      ;ENDFOLD
      ;FOLD -- RSK Fehlerausgabe KF1 Initiator/Motor -- ;%{SE}%MKUKATPVW %CVW_COM %VCOMMENT %P 2:-- RSK Fehlerausgabe KF1 Initiator/Motor --, 3: VW_COMMENT
      ;ENDFOLD
      ;FOLD F322 = !F313 ;%{SE}%MKUKATPVW %CVW_SPS %VBOASG %P 2:F322 = !F313, 3: BOASG
         $FLAG[322] = NOT $FLAG[313]
      ;ENDFOLD
      ;FOLD -- Fraesfehler -- ;%{SE}%MKUKATPVW %CVW_COM %VCOMMENT %P 2:-- Fraesfehler --, 3: VW_COMMENT
      ;ENDFOLD
      ;FOLD F329 = F324 + F322 ;%{SE}%MKUKATPVW %CVW_SPS %VBOASG %P 2:F329 = F324 + F322, 3: BOASG
         $FLAG[329] = $FLAG[324] OR $FLAG[322]
      ;ENDFOLD
      ;FOLD -- Fraeser aus bei Fehler -- ;%{SE}%MKUKATPVW %CVW_COM %VCOMMENT %P 2:-- Fraeser aus bei Fehler --, 3: VW_COMMENT
      ;ENDFOLD
      ;FOLD A864 = !F329 ;%{SE}%MKUKATPVW %CVW_SPS %VBOASG %P 2:A864 = !F329, 3: BOASG
         $OUT[864] = NOT $FLAG[329]
      ;ENDFOLD
      ;FOLD -- Warte Fraesen fertig oder Timeout -- ;%{SE}%MKUKATPVW %CVW_COM %VCOMMENT %P 2:-- Warte Fraesen fertig oder Timeout --, 3: VW_COMMENT
      ;ENDFOLD
      ;FOLD Schritt 124 = (F79 & F98 + F78 & F94 & !F287 + T7) & A4039 ;%{SE}%MKUKATPVW %CVW_SPS %VST_CON %P 2:Schritt 124 = (F79 & F98 + F78 & F94 & !F287 + T7) & A4039, 3: ST_CON
         IF ($FLAG[79] AND $FLAG[98] OR $FLAG[78] AND $FLAG[94] AND NOT $FLAG[287] OR $TIMER_FLAG[7]) AND $OUT[4039] THEN
            PREVSTEP = $APP_INT[5]
            $APP_INT[5] = 124
         ENDIF
      ;ENDFOLD
      ;FOLD Schritt 124 = (F78 & F96 & F287 + T7) & A4039 ;%{SE}%MKUKATPVW %CVW_SPS %VST_CON %P 2:Schritt 124 = (F78 & F96 & F287 + T7) & A4039, 3: ST_CON
         IF ($FLAG[78] AND $FLAG[96] AND $FLAG[287] OR $TIMER_FLAG[7]) AND $OUT[4039] THEN
            PREVSTEP = $APP_INT[5]
            $APP_INT[5] = 124
         ENDIF
      ;ENDFOLD
   ;ENDFOLD
   ;FOLD SCHRITT 124 -- ROB STP1 SZ1 -- ;%{P}%MKUKATPVW,%CSTEP,%VST_NR,%P 1:SCHRITT, 2:124, 3: ROB STP1 SZ1
      ;FOLD ;%{H}
         Case 124
      ;ENDFOLD
      ;FOLD -- Hilfsflag SK Programmwechsel -- ;%{SE}%MKUKATPVW %CVW_COM %VCOMMENT %P 2:-- Hilfsflag SK Programmwechsel --, 3: VW_COMMENT
      ;ENDFOLD
      ;FOLD F334 = AUS ;%{SE}%MKUKATPVW %CVW_SPS %VBOASG %P 2:F334 = AUS, 3: BOASG
         $FLAG[334] = FALSE
      ;ENDFOLD
      ;FOLD -- KF1 runterfahren -- ;%{SE}%MKUKATPVW %CVW_COM %VCOMMENT %P 2:-- KF1 runterfahren --, 3: VW_COMMENT
      ;ENDFOLD
      ;FOLD A863 = AUS ;%{SE}%MKUKATPVW %CVW_SPS %VBOASG %P 2:A863 = AUS, 3: BOASG
         $OUT[863] = FALSE
      ;ENDFOLD
      ;FOLD -- Fraesfehler -- ;%{SE}%MKUKATPVW %CVW_COM %VCOMMENT %P 2:-- Fraesfehler --, 3: VW_COMMENT
      ;ENDFOLD
      ;FOLD F329 = T7 + F324 ;%{SE}%MKUKATPVW %CVW_SPS %VBOASG %P 2:F329 = T7 + F324, 3: BOASG
         $FLAG[329] = $TIMER_FLAG[7] OR $FLAG[324]
      ;ENDFOLD
      ;FOLD -- Hilfsflag Startfraesen -- ;%{SE}%MKUKATPVW %CVW_COM %VCOMMENT %P 2:-- Hilfsflag Startfraesen --, 3: VW_COMMENT
      ;ENDFOLD
      ;FOLD F96 = F96 & F287 ;%{SE}%MKUKATPVW %CVW_SPS %VBOASG %P 2:F96 = F96 & F287, 3: BOASG
         $FLAG[96] = $FLAG[96] AND $FLAG[287]
      ;ENDFOLD
      ;FOLD F287 = F78 ;%{SE}%MKUKATPVW %CVW_SPS %VBOASG %P 2:F287 = F78, 3: BOASG
         $FLAG[287] = $FLAG[78]
      ;ENDFOLD
      ;FOLD -- Wiederholung beim Startfraesen -- ;%{SE}%MKUKATPVW %CVW_COM %VCOMMENT %P 2:-- Wiederholung beim Startfraesen --, 3: VW_COMMENT
      ;ENDFOLD
      ;FOLD Schritt 121 = E863 & F78 & !F96 & !F329 & A4039 ;%{SE}%MKUKATPVW %CVW_SPS %VST_CON %P 2:Schritt 121 = E863 & F78 & !F96 & !F329 & A4039, 3: ST_CON
         IF $IN[863] AND $FLAG[78] AND NOT $FLAG[96] AND NOT $FLAG[329] AND $OUT[4039] THEN
            PREVSTEP = $APP_INT[5]
            $APP_INT[5] = 121
         ENDIF
      ;ENDFOLD
      ;FOLD -- Weiter wenn Fraesen fertig -- ;%{SE}%MKUKATPVW %CVW_COM %VCOMMENT %P 2:-- Weiter wenn Fraesen fertig --, 3: VW_COMMENT
      ;ENDFOLD
      ;FOLD Schritt 125 = E863 & (F79 & F98 + F78 & F96 + F329) & A4039 ;%{SE}%MKUKATPVW %CVW_SPS %VST_CON %P 2:Schritt 125 = E863 & (F79 & F98 + F78 & F96 + F329) & A4039, 3: ST_CON
         IF $IN[863] AND ($FLAG[79] AND $FLAG[98] OR $FLAG[78] AND $FLAG[96] OR $FLAG[329]) AND $OUT[4039] THEN
            PREVSTEP = $APP_INT[5]
            $APP_INT[5] = 125
         ENDIF
      ;ENDFOLD
      ;FOLD -- Weiter bei Fehler -- ;%{SE}%MKUKATPVW %CVW_COM %VCOMMENT %P 2:-- Weiter bei Fehler --, 3: VW_COMMENT
      ;ENDFOLD
      ;FOLD Schritt 127 = F329 & (E26 + E27) & A4039 ;%{SE}%MKUKATPVW %CVW_SPS %VST_CON %P 2:Schritt 127 = F329 & (E26 + E27) & A4039, 3: ST_CON
         IF $FLAG[329] AND ($IN[26] OR $IN[27]) AND $OUT[4039] THEN
            PREVSTEP = $APP_INT[5]
            $APP_INT[5] = 127
         ENDIF
      ;ENDFOLD
   ;ENDFOLD
   ;FOLD SCHRITT 125 -- ROB STP1 SZ1 -- ;%{P}%MKUKATPVW,%CSTEP,%VST_NR,%P 1:SCHRITT, 2:125, 3: ROB STP1 SZ1
      ;FOLD ;%{H}
         Case 125
      ;ENDFOLD
      ;FOLD -- KF1 einschalten -- ;%{SE}%MKUKATPVW %CVW_COM %VCOMMENT %P 2:-- KF1 einschalten --, 3: VW_COMMENT
      ;ENDFOLD
      ;FOLD A864 = AUS ;%{SE}%MKUKATPVW %CVW_SPS %VBOASG %P 2:A864 = AUS, 3: BOASG
         $OUT[864] = FALSE
      ;ENDFOLD
      ;FOLD bin3 (!F329) = 1 ;%{SE}%MKUKATPVW %CVW_SPS %VARIASG %P 2:bin3 (!F329) = 1, 3: ARIASG
         VW(#BINOUT,NOT $FLAG[329],3,1)
      ;ENDFOLD
      ;FOLD -- Wartezeit Programmwechsel SK -- ;%{SE}%MKUKATPVW %CVW_COM %VCOMMENT %P 2:-- Wartezeit Programmwechsel SK --, 3: VW_COMMENT
      ;ENDFOLD
      ;FOLD T8 ( !F334 ) = -2[1/10Sek] ;%{SE}%MKUKATPVW %CVW_SPS %VTASG %P 2:T8 ( !F334 ) = -2[1/10Sek], 3: TASG
         VW(#SET_TIME,NOT $FLAG[334],8,0,-2)
      ;ENDFOLD
      ;FOLD -- Hilfsflag SK Programmwechsel -- ;%{SE}%MKUKATPVW %CVW_COM %VCOMMENT %P 2:-- Hilfsflag SK Programmwechsel --, 3: VW_COMMENT
      ;ENDFOLD
      ;FOLD F334 = EIN ;%{SE}%MKUKATPVW %CVW_SPS %VBOASG %P 2:F334 = EIN, 3: BOASG
         $FLAG[334] = TRUE
      ;ENDFOLD
      ;FOLD Schritt 126 = T8 & A4039 ;%{SE}%MKUKATPVW %CVW_SPS %VST_CON %P 2:Schritt 126 = T8 & A4039, 3: ST_CON
         IF $TIMER_FLAG[8] AND $OUT[4039] THEN
            PREVSTEP = $APP_INT[5]
            $APP_INT[5] = 126
         ENDIF
      ;ENDFOLD
   ;ENDFOLD
   ;FOLD SCHRITT 126 -- ROB STP1 SZ1 -- ;%{P}%MKUKATPVW,%CSTEP,%VST_NR,%P 1:SCHRITT, 2:126, 3: ROB STP1 SZ1
      ;FOLD ;%{H}
         Case 126
      ;ENDFOLD
      ;FOLD -- Hilfsflag SK Programmwechsel -- ;%{SE}%MKUKATPVW %CVW_COM %VCOMMENT %P 2:-- Hilfsflag SK Programmwechsel --, 3: VW_COMMENT
      ;ENDFOLD
      ;FOLD F334 = AUS ;%{SE}%MKUKATPVW %CVW_SPS %VBOASG %P 2:F334 = AUS, 3: BOASG
         $FLAG[334] = FALSE
      ;ENDFOLD
      ;FOLD -- RSK Sammelstoerung -- ;%{SE}%MKUKATPVW %CVW_COM %VCOMMENT %P 2:-- RSK Sammelstoerung --, 3: VW_COMMENT
      ;ENDFOLD
      ;FOLD F329 = T7 ;%{SE}%MKUKATPVW %CVW_SPS %VBOASG %P 2:F329 = T7, 3: BOASG
         $FLAG[329] = $TIMER_FLAG[7]
      ;ENDFOLD
      ;FOLD -- Quitt. Fraesen SK1 -- ;%{SE}%MKUKATPVW %CVW_COM %VCOMMENT %P 2:-- Quitt. Fraesen SK1 --, 3: VW_COMMENT
      ;ENDFOLD
      ;FOLD A786 = !F329 & !F322 ;%{SE}%MKUKATPVW %CVW_SPS %VBOASG %P 2:A786 = !F329 & !F322, 3: BOASG
         $OUT[786] = NOT $FLAG[329] AND NOT $FLAG[322]
      ;ENDFOLD
      ;FOLD Schritt 127 = !E786 & E787 & !E788 & !F329 ;%{SE}%MKUKATPVW %CVW_SPS %VST_CON %P 2:Schritt 127 = !E786 & E787 & !E788 & !F329, 3: ST_CON
         IF NOT $IN[786] AND $IN[787] AND NOT $IN[788] AND NOT $FLAG[329] THEN
            PREVSTEP = $APP_INT[5]
            $APP_INT[5] = 127
         ENDIF
      ;ENDFOLD
   ;ENDFOLD
   ;FOLD SCHRITT 127 -- ROB STP1 SZ1 # Ende -- ;%{P}%MKUKATPVW,%CSTEP,%VST_NR,%P 1:SCHRITT, 2:127, 3: ROB STP1 SZ1 # Ende
      ;FOLD ;%{H}
         Case 127
      ;ENDFOLD
      ;FOLD -- RSK Sammelstoerung -- ;%{SE}%MKUKATPVW %CVW_COM %VCOMMENT %P 2:-- RSK Sammelstoerung --, 3: VW_COMMENT
      ;ENDFOLD
      ;FOLD F329 = T7 ;%{SE}%MKUKATPVW %CVW_SPS %VBOASG %P 2:F329 = T7, 3: BOASG
         $FLAG[329] = $TIMER_FLAG[7]
      ;ENDFOLD
      ;FOLD F91 = !F329 ;%{SE}%MKUKATPVW %CVW_SPS %VBOASG %P 2:F91 = !F329, 3: BOASG
         $FLAG[91] = NOT $FLAG[329]
      ;ENDFOLD
      ;FOLD Schritt 120 = F329 & (E26 + E27) & A4039 ;%{SE}%MKUKATPVW %CVW_SPS %VST_CON %P 2:Schritt 120 = F329 & (E26 + E27) & A4039, 3: ST_CON
         IF $FLAG[329] AND ($IN[26] OR $IN[27]) AND $OUT[4039] THEN
            PREVSTEP = $APP_INT[5]
            $APP_INT[5] = 120
         ENDIF
      ;ENDFOLD
      ;FOLD Schritt 1 = F91 & !F329 & A4039 ;%{SE}%MKUKATPVW %CVW_SPS %VST_CON %P 2:Schritt 1 = F91 & !F329 & A4039, 3: ST_CON
         IF $FLAG[91] AND NOT $FLAG[329] AND $OUT[4039] THEN
            PREVSTEP = $APP_INT[5]
            $APP_INT[5] = 1
         ENDIF
      ;ENDFOLD
   ;ENDFOLD
   ;FOLD SCHRITT 128 -- MS1 Reinigung (an KS3)-- ;%{P}%MKUKATPVW,%CSTEP,%VST_NR,%P 1:SCHRITT, 2:128, 3: MS1 Reinigung (an KS3)
      ;FOLD ;%{H}
         Case 128
      ;ENDFOLD
      ;FOLD -- RSK gestartet -- ;%{SE}%MKUKATPVW %CVW_COM %VCOMMENT %P 2:-- RSK gestartet --, 3: VW_COMMENT
      ;ENDFOLD
      ;FOLD F321 = AUS ;%{SE}%MKUKATPVW %CVW_SPS %VBOASG %P 2:F321 = AUS, 3: BOASG
         $FLAG[321] = FALSE
      ;ENDFOLD
      ;FOLD F323 = AUS ;%{SE}%MKUKATPVW %CVW_SPS %VBOASG %P 2:F323 = AUS, 3: BOASG
         $FLAG[323] = FALSE
      ;ENDFOLD
      ;FOLD F324 = AUS ;%{SE}%MKUKATPVW %CVW_SPS %VBOASG %P 2:F324 = AUS, 3: BOASG
         $FLAG[324] = FALSE
      ;ENDFOLD
      ;FOLD F329 = AUS ;%{SE}%MKUKATPVW %CVW_SPS %VBOASG %P 2:F329 = AUS, 3: BOASG
         $FLAG[329] = FALSE
      ;ENDFOLD
      ;FOLD -- MS1 Reinigung gestartet -- ;%{SE}%MKUKATPVW %CVW_COM %VCOMMENT %P 2:-- MS1 Reinigung gestartet --, 3: VW_COMMENT
      ;ENDFOLD
      ;FOLD F604 = EIN ;%{SE}%MKUKATPVW %CVW_SPS %VBOASG %P 2:F604 = EIN, 3: BOASG
         $FLAG[604] = TRUE
      ;ENDFOLD
      ;FOLD -- Ueberwachungszeit KS3 schwenken -- ;%{SE}%MKUKATPVW %CVW_COM %VCOMMENT %P 2:-- Ueberwachungszeit KS3 schwenken --, 3: VW_COMMENT
      ;ENDFOLD
      ;FOLD t8 ( EIN ) = -100[1/10Sek] ;%{SE}%MKUKATPVW %CVW_SPS %VTASG %P 2:t8 ( EIN ) = -100[1/10Sek], 3: TASG
         VW(#SET_TIME,TRUE,8,0,-100)
      ;ENDFOLD
      ;FOLD Schritt 129 = A4039 ;%{SE}%MKUKATPVW %CVW_SPS %VST_CON %P 2:Schritt 129 = A4039, 3: ST_CON
         IF $OUT[4039] THEN
            PREVSTEP = $APP_INT[5]
            $APP_INT[5] = 129
         ENDIF
      ;ENDFOLD
   ;ENDFOLD
   ;FOLD SCHRITT 129 -- MS1 Reinigung (an KS3) -- ;%{P}%MKUKATPVW,%CSTEP,%VST_NR,%P 1:SCHRITT, 2:129, 3: MS1 Reinigung (an KS3)
      ;FOLD ;%{H}
         Case 129
      ;ENDFOLD
      ;FOLD -- RSK Fehlerausgabe KS3 Ruhest. -- ;%{SE}%MKUKATPVW %CVW_COM %VCOMMENT %P 2:-- RSK Fehlerausgabe KS3 Ruhest. --, 3: VW_COMMENT
      ;ENDFOLD
      ;FOLD F323 = !E1156 ;%{SE}%MKUKATPVW %CVW_SPS %VBOASG %P 2:F323 = !E1156, 3: BOASG
         $FLAG[323] = NOT $IN[1156]
      ;ENDFOLD
      ;FOLD -- RSK Sammelstoerung -- ;%{SE}%MKUKATPVW %CVW_COM %VCOMMENT %P 2:-- RSK Sammelstoerung --, 3: VW_COMMENT
      ;ENDFOLD
      ;FOLD F329 = F323 ;%{SE}%MKUKATPVW %CVW_SPS %VBOASG %P 2:F329 = F323, 3: BOASG
         $FLAG[329] = $FLAG[323]
      ;ENDFOLD
      ;FOLD Schritt 128 = (E26 + E27) & F323 & A4039 ;%{SE}%MKUKATPVW %CVW_SPS %VST_CON %P 2:Schritt 128 = (E26 + E27) & F323 & A4039, 3: ST_CON
         IF ($IN[26] OR $IN[27]) AND $FLAG[323] AND $OUT[4039] THEN
            PREVSTEP = $APP_INT[5]
            $APP_INT[5] = 128
         ENDIF
      ;ENDFOLD
      ;FOLD Schritt 130 = (!F323 + T8) & A4039 ;%{SE}%MKUKATPVW %CVW_SPS %VST_CON %P 2:Schritt 130 = (!F323 + T8) & A4039, 3: ST_CON
         IF (NOT $FLAG[323] OR $TIMER_FLAG[8]) AND $OUT[4039] THEN
            PREVSTEP = $APP_INT[5]
            $APP_INT[5] = 130
         ENDIF
      ;ENDFOLD
   ;ENDFOLD
   ;FOLD SCHRITT 130 -- MS1 Reinigung (an KS3) -- ;%{P}%MKUKATPVW,%CSTEP,%VST_NR,%P 1:SCHRITT, 2:130, 3: MS1 Reinigung (an KS3)
      ;FOLD ;%{H}
         Case 130
      ;ENDFOLD
      ;FOLD -- KS3 in Arbeitsstellung schwenken -- ;%{SE}%MKUKATPVW %CVW_COM %VCOMMENT %P 2:-- KS3 in Arbeitsstellung schwenken --, 3: VW_COMMENT
      ;ENDFOLD
      ;FOLD A1160 = !E1157 ;%{SE}%MKUKATPVW %CVW_SPS %VBOASG %P 2:A1160 = !E1157, 3: BOASG
         $OUT[1160] = NOT $IN[1157]
      ;ENDFOLD
      ;FOLD Schritt 131 = A4039 ;%{SE}%MKUKATPVW %CVW_SPS %VST_CON %P 2:Schritt 131 = A4039, 3: ST_CON
         IF $OUT[4039] THEN
            PREVSTEP = $APP_INT[5]
            $APP_INT[5] = 131
         ENDIF
      ;ENDFOLD
   ;ENDFOLD
   ;FOLD SCHRITT 131 -- MS1 Reinigung (an KS3) -- ;%{P}%MKUKATPVW,%CSTEP,%VST_NR,%P 1:SCHRITT, 2:131, 3: MS1 Reinigung (an KS3)
      ;FOLD ;%{H}
         Case 131
      ;ENDFOLD
      ;FOLD -- RSK Fehlerausgabe KS3 Arbeitsstellung -- ;%{SE}%MKUKATPVW %CVW_COM %VCOMMENT %P 2:-- RSK Fehlerausgabe KS3 Arbeitsstellung --, 3: VW_COMMENT
      ;ENDFOLD
      ;FOLD F324 = !E1157 & T8 + F324 ;%{SE}%MKUKATPVW %CVW_SPS %VBOASG %P 2:F324 = !E1157 & T8 + F324, 3: BOASG
         $FLAG[324] = NOT $IN[1157] AND $TIMER_FLAG[8] OR $FLAG[324]
      ;ENDFOLD
      ;FOLD -- RSK Sammelstoerung -- ;%{SE}%MKUKATPVW %CVW_COM %VCOMMENT %P 2:-- RSK Sammelstoerung --, 3: VW_COMMENT
      ;ENDFOLD
      ;FOLD F329 = F324 ;%{SE}%MKUKATPVW %CVW_SPS %VBOASG %P 2:F329 = F324, 3: BOASG
         $FLAG[329] = $FLAG[324]
      ;ENDFOLD
      ;FOLD Schritt 128 = F324 & (E26 + E27) & A4039 ;%{SE}%MKUKATPVW %CVW_SPS %VST_CON %P 2:Schritt 128 = F324 & (E26 + E27) & A4039, 3: ST_CON
         IF $FLAG[324] AND ($IN[26] OR $IN[27]) AND $OUT[4039] THEN
            PREVSTEP = $APP_INT[5]
            $APP_INT[5] = 128
         ENDIF
      ;ENDFOLD
      ;FOLD Schritt 132 = !F324 & E1157 & !E1159 & A4039 ;%{SE}%MKUKATPVW %CVW_SPS %VST_CON %P 2:Schritt 132 = !F324 & E1157 & !E1159 & A4039, 3: ST_CON
         IF NOT $FLAG[324] AND $IN[1157] AND NOT $IN[1159] AND $OUT[4039] THEN
            PREVSTEP = $APP_INT[5]
            $APP_INT[5] = 132
         ENDIF
      ;ENDFOLD
   ;ENDFOLD
   ;FOLD SCHRITT 132 -- MS1 Reinigung (an KS3) -- ;%{P}%MKUKATPVW,%CSTEP,%VST_NR,%P 1:SCHRITT, 2:132, 3: MS1 Reinigung (an KS3)
      ;FOLD ;%{H}
         Case 132
      ;ENDFOLD
      ;FOLD A1864 = AUS ;%{SE}%MKUKATPVW %CVW_SPS %VBOASG %P 2:A1864 = AUS, 3: BOASG
         $OUT[1864] = FALSE
      ;ENDFOLD
      ;FOLD A2168 = AUS ;%{SE}%MKUKATPVW %CVW_SPS %VBOASG %P 2:A2168 = AUS, 3: BOASG
         $OUT[2168] = FALSE
      ;ENDFOLD
      ;FOLD -- Ueberwachungszeit Versetzeinheit -- ;%{SE}%MKUKATPVW %CVW_COM %VCOMMENT %P 2:-- Ueberwachungszeit Versetzeinheit --, 3: VW_COMMENT
      ;ENDFOLD
      ;FOLD t8 ( EIN ) = -50[1/10Sek] ;%{SE}%MKUKATPVW %CVW_SPS %VTASG %P 2:t8 ( EIN ) = -50[1/10Sek], 3: TASG
         VW(#SET_TIME,TRUE,8,0,-50)
      ;ENDFOLD
      ;FOLD -- Ueberwachungszeit Reinigung -- ;%{SE}%MKUKATPVW %CVW_COM %VCOMMENT %P 2:-- Ueberwachungszeit Reinigung --, 3: VW_COMMENT
      ;ENDFOLD
      ;FOLD t9 ( EIN ) = -80[1/10Sek] ;%{SE}%MKUKATPVW %CVW_SPS %VTASG %P 2:t9 ( EIN ) = -80[1/10Sek], 3: TASG
         VW(#SET_TIME,TRUE,9,0,-80)
      ;ENDFOLD
      ;FOLD Schritt 133 = A4039 ;%{SE}%MKUKATPVW %CVW_SPS %VST_CON %P 2:Schritt 133 = A4039, 3: ST_CON
         IF $OUT[4039] THEN
            PREVSTEP = $APP_INT[5]
            $APP_INT[5] = 133
         ENDIF
      ;ENDFOLD
   ;ENDFOLD
   ;FOLD SCHRITT 133 -- MS1 Reinigung (an KS3) -- ;%{P}%MKUKATPVW,%CSTEP,%VST_NR,%P 1:SCHRITT, 2:133, 3: MS1 Reinigung (an KS3)
      ;FOLD ;%{H}
         Case 133
      ;ENDFOLD
      ;FOLD -- RSK Fehlerausgabe Versetzeinheit -- ;%{SE}%MKUKATPVW %CVW_COM %VCOMMENT %P 2:-- RSK Fehlerausgabe Versetzeinheit --, 3: VW_COMMENT
      ;ENDFOLD
      ;FOLD F328 = F576 & T8 ;%{SE}%MKUKATPVW %CVW_SPS %VBOASG %P 2:F328 = F576 & T8, 3: BOASG
         $FLAG[328] = $FLAG[576] AND $TIMER_FLAG[8]
      ;ENDFOLD
      ;FOLD -- RSK Sammelstoerung -- ;%{SE}%MKUKATPVW %CVW_COM %VCOMMENT %P 2:-- RSK Sammelstoerung --, 3: VW_COMMENT
      ;ENDFOLD
      ;FOLD F329 = T8 ;%{SE}%MKUKATPVW %CVW_SPS %VBOASG %P 2:F329 = T8, 3: BOASG
         $FLAG[329] = $TIMER_FLAG[8]
      ;ENDFOLD
      ;FOLD -- Versetzeinheit in Arbeitsst. schw. -- ;%{SE}%MKUKATPVW %CVW_COM %VCOMMENT %P 2:-- Versetzeinheit in Arbeitsst. schw. --, 3: VW_COMMENT
      ;ENDFOLD
      ;FOLD A2168 = !E2168 & F576 ;%{SE}%MKUKATPVW %CVW_SPS %VBOASG %P 2:A2168 = !E2168 & F576, 3: BOASG
         $OUT[2168] = NOT $IN[2168] AND $FLAG[576]
      ;ENDFOLD
      ;FOLD Schritt 132 = A2168 & T8 & (E26 + E27) & A4039 ;%{SE}%MKUKATPVW %CVW_SPS %VST_CON %P 2:Schritt 132 = A2168 & T8 & (E26 + E27) & A4039, 3: ST_CON
         IF $OUT[2168] AND $TIMER_FLAG[8] AND ($IN[26] OR $IN[27]) AND $OUT[4039] THEN
            PREVSTEP = $APP_INT[5]
            $APP_INT[5] = 132
         ENDIF
      ;ENDFOLD
      ;FOLD Schritt 134 = (E2168 & F576 + !E2168 & !F576) & A4039 ;%{SE}%MKUKATPVW %CVW_SPS %VST_CON %P 2:Schritt 134 = (E2168 & F576 + !E2168 & !F576) & A4039, 3: ST_CON
         IF ($IN[2168] AND $FLAG[576] OR NOT $IN[2168] AND NOT $FLAG[576]) AND $OUT[4039] THEN
            PREVSTEP = $APP_INT[5]
            $APP_INT[5] = 134
         ENDIF
      ;ENDFOLD
   ;ENDFOLD
   ;FOLD SCHRITT 134 -- MS1 Reinigung (an KS3) -- ;%{P}%MKUKATPVW,%CSTEP,%VST_NR,%P 1:SCHRITT, 2:134, 3: MS1 Reinigung (an KS3)
      ;FOLD ;%{H}
         Case 134
      ;ENDFOLD
      ;FOLD -- RSK Sammelstoerung -- ;%{SE}%MKUKATPVW %CVW_COM %VCOMMENT %P 2:-- RSK Sammelstoerung --, 3: VW_COMMENT
      ;ENDFOLD
      ;FOLD F329 = T9 ;%{SE}%MKUKATPVW %CVW_SPS %VBOASG %P 2:F329 = T9, 3: BOASG
         $FLAG[329] = $TIMER_FLAG[9]
      ;ENDFOLD
      ;FOLD -- MS1 Ausblasen EIN -- ;%{SE}%MKUKATPVW %CVW_COM %VCOMMENT %P 2:-- MS1 Ausblasen EIN --, 3: VW_COMMENT
      ;ENDFOLD
      ;FOLD A1870 = EIN ;%{SE}%MKUKATPVW %CVW_SPS %VBOASG %P 2:A1870 = EIN, 3: BOASG
         $OUT[1870] = TRUE
      ;ENDFOLD
      ;FOLD -- MS1 Reinigung starten -- ;%{SE}%MKUKATPVW %CVW_COM %VCOMMENT %P 2:-- MS1 Reinigung starten --, 3: VW_COMMENT
      ;ENDFOLD
      ;FOLD A1864 = EIN ;%{SE}%MKUKATPVW %CVW_SPS %VBOASG %P 2:A1864 = EIN, 3: BOASG
         $OUT[1864] = TRUE
      ;ENDFOLD
      ;FOLD Schritt 132 = !E1864 & T9 & (E26 + E27) & A4039 ;%{SE}%MKUKATPVW %CVW_SPS %VST_CON %P 2:Schritt 132 = !E1864 & T9 & (E26 + E27) & A4039, 3: ST_CON
         IF NOT $IN[1864] AND $TIMER_FLAG[9] AND ($IN[26] OR $IN[27]) AND $OUT[4039] THEN
            PREVSTEP = $APP_INT[5]
            $APP_INT[5] = 132
         ENDIF
      ;ENDFOLD
      ;FOLD Schritt 135 = E1864 & A4039 ;%{SE}%MKUKATPVW %CVW_SPS %VST_CON %P 2:Schritt 135 = E1864 & A4039, 3: ST_CON
         IF $IN[1864] AND $OUT[4039] THEN
            PREVSTEP = $APP_INT[5]
            $APP_INT[5] = 135
         ENDIF
      ;ENDFOLD
   ;ENDFOLD
   ;FOLD SCHRITT 135 -- MS1 Reinigung (an KS3) -- ;%{P}%MKUKATPVW,%CSTEP,%VST_NR,%P 1:SCHRITT, 2:135, 3: MS1 Reinigung (an KS3)
      ;FOLD ;%{H}
         Case 135
      ;ENDFOLD
      ;FOLD -- MS1 Reinigung beenden -- ;%{SE}%MKUKATPVW %CVW_COM %VCOMMENT %P 2:-- MS1 Reinigung beenden --, 3: VW_COMMENT
      ;ENDFOLD
      ;FOLD A1864 = AUS ;%{SE}%MKUKATPVW %CVW_SPS %VBOASG %P 2:A1864 = AUS, 3: BOASG
         $OUT[1864] = FALSE
      ;ENDFOLD
      ;FOLD -- MS1 Ausblasen AUS -- ;%{SE}%MKUKATPVW %CVW_COM %VCOMMENT %P 2:-- MS1 Ausblasen AUS --, 3: VW_COMMENT
      ;ENDFOLD
      ;FOLD A1870 = AUS ;%{SE}%MKUKATPVW %CVW_SPS %VBOASG %P 2:A1870 = AUS, 3: BOASG
         $OUT[1870] = FALSE
      ;ENDFOLD
      ;FOLD -- MS1 Einspruehen EIN -- ;%{SE}%MKUKATPVW %CVW_COM %VCOMMENT %P 2:-- MS1 Einspruehen EIN --, 3: VW_COMMENT
      ;ENDFOLD
      ;FOLD A520 = !F574 & F575 ;%{SE}%MKUKATPVW %CVW_SPS %VBOASG %P 2:A520 = !F574 & F575, 3: BOASG
         $OUT[520] = NOT $FLAG[574] AND $FLAG[575]
      ;ENDFOLD
      ;FOLD A1871 = F574 & F575 ;%{SE}%MKUKATPVW %CVW_SPS %VBOASG %P 2:A1871 = F574 & F575, 3: BOASG
         $OUT[1871] = $FLAG[574] AND $FLAG[575]
      ;ENDFOLD
      ;FOLD -- Einschaltdauer Einspruehen -- ;%{SE}%MKUKATPVW %CVW_COM %VCOMMENT %P 2:-- Einschaltdauer Einspruehen --, 3: VW_COMMENT
      ;ENDFOLD
      ;FOLD t7 ( EIN ) = i23[1/10Sek] ;%{SE}%MKUKATPVW %CVW_SPS %VTASG %P 2:t7 ( EIN ) = i23[1/10Sek], 3: TASG
         VW(#SET_TIME,TRUE,7,0,$COUNT_I[23])
      ;ENDFOLD
      ;FOLD Schritt 136 = A4039 ;%{SE}%MKUKATPVW %CVW_SPS %VST_CON %P 2:Schritt 136 = A4039, 3: ST_CON
         IF $OUT[4039] THEN
            PREVSTEP = $APP_INT[5]
            $APP_INT[5] = 136
         ENDIF
      ;ENDFOLD
   ;ENDFOLD
   ;FOLD SCHRITT 136 -- MS1 Reinigung (an KS3) -- ;%{P}%MKUKATPVW,%CSTEP,%VST_NR,%P 1:SCHRITT, 2:136, 3: MS1 Reinigung (an KS3)
      ;FOLD ;%{H}
         Case 136
      ;ENDFOLD
      ;FOLD F323 = AUS ;%{SE}%MKUKATPVW %CVW_SPS %VBOASG %P 2:F323 = AUS, 3: BOASG
         $FLAG[323] = FALSE
      ;ENDFOLD
      ;FOLD -- Ueberwachungszeit KS3 schwenken -- ;%{SE}%MKUKATPVW %CVW_COM %VCOMMENT %P 2:-- Ueberwachungszeit KS3 schwenken --, 3: VW_COMMENT
      ;ENDFOLD
      ;FOLD t8 ( EIN ) = -100[1/10Sek] ;%{SE}%MKUKATPVW %CVW_SPS %VTASG %P 2:t8 ( EIN ) = -100[1/10Sek], 3: TASG
         VW(#SET_TIME,TRUE,8,0,-100)
      ;ENDFOLD
      ;FOLD Schritt 137 = T7 & A4039 ;%{SE}%MKUKATPVW %CVW_SPS %VST_CON %P 2:Schritt 137 = T7 & A4039, 3: ST_CON
         IF $TIMER_FLAG[7] AND $OUT[4039] THEN
            PREVSTEP = $APP_INT[5]
            $APP_INT[5] = 137
         ENDIF
      ;ENDFOLD
   ;ENDFOLD
   ;FOLD SCHRITT 137 -- MS1 Reinigung (an KS3) -- ;%{P}%MKUKATPVW,%CSTEP,%VST_NR,%P 1:SCHRITT, 2:137, 3: MS1 Reinigung (an KS3)
      ;FOLD ;%{H}
         Case 137
      ;ENDFOLD
      ;FOLD -- MS1 Einspruehen AUS -- ;%{SE}%MKUKATPVW %CVW_COM %VCOMMENT %P 2:-- MS1 Einspruehen AUS --, 3: VW_COMMENT
      ;ENDFOLD
      ;FOLD A520 = AUS ;%{SE}%MKUKATPVW %CVW_SPS %VBOASG %P 2:A520 = AUS, 3: BOASG
         $OUT[520] = FALSE
      ;ENDFOLD
      ;FOLD A1871 = AUS ;%{SE}%MKUKATPVW %CVW_SPS %VBOASG %P 2:A1871 = AUS, 3: BOASG
         $OUT[1871] = FALSE
      ;ENDFOLD
      ;FOLD -- RSK Fehlerausgabe KS3 Ruhest. -- ;%{SE}%MKUKATPVW %CVW_COM %VCOMMENT %P 2:-- RSK Fehlerausgabe KS3 Ruhest. --, 3: VW_COMMENT
      ;ENDFOLD
      ;FOLD F324 = !E1157 ;%{SE}%MKUKATPVW %CVW_SPS %VBOASG %P 2:F324 = !E1157, 3: BOASG
         $FLAG[324] = NOT $IN[1157]
      ;ENDFOLD
      ;FOLD -- RSK Sammelstoerung -- ;%{SE}%MKUKATPVW %CVW_COM %VCOMMENT %P 2:-- RSK Sammelstoerung --, 3: VW_COMMENT
      ;ENDFOLD
      ;FOLD F329 = F324 + T8 ;%{SE}%MKUKATPVW %CVW_SPS %VBOASG %P 2:F329 = F324 + T8, 3: BOASG
         $FLAG[329] = $FLAG[324] OR $TIMER_FLAG[8]
      ;ENDFOLD
      ;FOLD Schritt 136 = (E26 + E27) & F324 & A4039 ;%{SE}%MKUKATPVW %CVW_SPS %VST_CON %P 2:Schritt 136 = (E26 + E27) & F324 & A4039, 3: ST_CON
         IF ($IN[26] OR $IN[27]) AND $FLAG[324] AND $OUT[4039] THEN
            PREVSTEP = $APP_INT[5]
            $APP_INT[5] = 136
         ENDIF
      ;ENDFOLD
      ;FOLD Schritt 138 = (!F324 + T8) & A4039 ;%{SE}%MKUKATPVW %CVW_SPS %VST_CON %P 2:Schritt 138 = (!F324 + T8) & A4039, 3: ST_CON
         IF (NOT $FLAG[324] OR $TIMER_FLAG[8]) AND $OUT[4039] THEN
            PREVSTEP = $APP_INT[5]
            $APP_INT[5] = 138
         ENDIF
      ;ENDFOLD
   ;ENDFOLD
   ;FOLD SCHRITT 138 -- MS1 Reinigung (an KS3) -- ;%{P}%MKUKATPVW,%CSTEP,%VST_NR,%P 1:SCHRITT, 2:138, 3: MS1 Reinigung (an KS3)
      ;FOLD ;%{H}
         Case 138
      ;ENDFOLD
      ;FOLD -- KS3 in Ruhestellung schwenken -- ;%{SE}%MKUKATPVW %CVW_COM %VCOMMENT %P 2:-- KS3 in Ruhestellung schwenken --, 3: VW_COMMENT
      ;ENDFOLD
      ;FOLD A1160 = !E1156 ;%{SE}%MKUKATPVW %CVW_SPS %VBOASG %P 2:A1160 = !E1156, 3: BOASG
         $OUT[1160] = NOT $IN[1156]
      ;ENDFOLD
      ;FOLD Schritt 139 = A4039 ;%{SE}%MKUKATPVW %CVW_SPS %VST_CON %P 2:Schritt 139 = A4039, 3: ST_CON
         IF $OUT[4039] THEN
            PREVSTEP = $APP_INT[5]
            $APP_INT[5] = 139
         ENDIF
      ;ENDFOLD
   ;ENDFOLD
   ;FOLD SCHRITT 139 -- MS1 Reinigung (an KS3) -- ;%{P}%MKUKATPVW,%CSTEP,%VST_NR,%P 1:SCHRITT, 2:139, 3: MS1 Reinigung (an KS3)
      ;FOLD ;%{H}
         Case 139
      ;ENDFOLD
      ;FOLD -- RSK Fehlerausgabe KS3 Ruhestellung -- ;%{SE}%MKUKATPVW %CVW_COM %VCOMMENT %P 2:-- RSK Fehlerausgabe KS3 Ruhestellung --, 3: VW_COMMENT
      ;ENDFOLD
      ;FOLD F323 = !E1156 & T8 + F323 ;%{SE}%MKUKATPVW %CVW_SPS %VBOASG %P 2:F323 = !E1156 & T8 + F323, 3: BOASG
         $FLAG[323] = NOT $IN[1156] AND $TIMER_FLAG[8] OR $FLAG[323]
      ;ENDFOLD
      ;FOLD -- RSK Sammelstoerung -- ;%{SE}%MKUKATPVW %CVW_COM %VCOMMENT %P 2:-- RSK Sammelstoerung --, 3: VW_COMMENT
      ;ENDFOLD
      ;FOLD F329 = F323 ;%{SE}%MKUKATPVW %CVW_SPS %VBOASG %P 2:F329 = F323, 3: BOASG
         $FLAG[329] = $FLAG[323]
      ;ENDFOLD
      ;FOLD Schritt 136 = F323 & (E26 + E27) & A4039 ;%{SE}%MKUKATPVW %CVW_SPS %VST_CON %P 2:Schritt 136 = F323 & (E26 + E27) & A4039, 3: ST_CON
         IF $FLAG[323] AND ($IN[26] OR $IN[27]) AND $OUT[4039] THEN
            PREVSTEP = $APP_INT[5]
            $APP_INT[5] = 136
         ENDIF
      ;ENDFOLD
      ;FOLD Schritt 140 = E1156 & !E1158 & A4039 ;%{SE}%MKUKATPVW %CVW_SPS %VST_CON %P 2:Schritt 140 = E1156 & !E1158 & A4039, 3: ST_CON
         IF $IN[1156] AND NOT $IN[1158] AND $OUT[4039] THEN
            PREVSTEP = $APP_INT[5]
            $APP_INT[5] = 140
         ENDIF
      ;ENDFOLD
   ;ENDFOLD
   ;FOLD SCHRITT 140 -- MS1 Reinigung (an KS3) -- ;%{P}%MKUKATPVW,%CSTEP,%VST_NR,%P 1:SCHRITT, 2:140, 3: MS1 Reinigung (an KS3)
      ;FOLD ;%{H}
         Case 140
      ;ENDFOLD
      ;FOLD F323 = AUS ;%{SE}%MKUKATPVW %CVW_SPS %VBOASG %P 2:F323 = AUS, 3: BOASG
         $FLAG[323] = FALSE
      ;ENDFOLD
      ;FOLD F329 = AUS ;%{SE}%MKUKATPVW %CVW_SPS %VBOASG %P 2:F329 = AUS, 3: BOASG
         $FLAG[329] = FALSE
      ;ENDFOLD
      ;FOLD -- MS1 Zaehler ruecksetzen -- ;%{SE}%MKUKATPVW %CVW_COM %VCOMMENT %P 2:-- MS1 Zaehler ruecksetzen --, 3: VW_COMMENT
      ;ENDFOLD
      ;FOLD -- MS1 FRG Reinigung -- ;%{SE}%MKUKATPVW %CVW_COM %VCOMMENT %P 2:-- MS1 FRG Reinigung --, 3: VW_COMMENT
      ;ENDFOLD
      ;FOLD F603 = AUS ;%{SE}%MKUKATPVW %CVW_SPS %VBOASG %P 2:F603 = AUS, 3: BOASG
         $FLAG[603] = FALSE
      ;ENDFOLD
      ;FOLD -- MS1 Reinigung FK -- ;%{SE}%MKUKATPVW %CVW_COM %VCOMMENT %P 2:-- MS1 Reinigung FK --, 3: VW_COMMENT
      ;ENDFOLD
      ;FOLD F605 = EIN ;%{SE}%MKUKATPVW %CVW_SPS %VBOASG %P 2:F605 = EIN, 3: BOASG
         $FLAG[605] = TRUE
      ;ENDFOLD
      ;FOLD t8 ( EIN ) = STOP ;%{SE}%MKUKATPVW %CVW_SPS %VTSTOP %P 2:t8 ( EIN ) = STOP, 3: TSTOP
         VW(#SET_TIME,TRUE,8,1,0)
      ;ENDFOLD
      ;FOLD Schritt 1 = A4039 ;%{SE}%MKUKATPVW %CVW_SPS %VST_CON %P 2:Schritt 1 = A4039, 3: ST_CON
         IF $OUT[4039] THEN
            PREVSTEP = $APP_INT[5]
            $APP_INT[5] = 1
         ENDIF
      ;ENDFOLD
   ;ENDFOLD
   ;FOLD SCHRITT 141 -- MS2 Reinigung (an KS2) -- ;%{P}%MKUKATPVW,%CSTEP,%VST_NR,%P 1:SCHRITT, 2:141, 3: MS2 Reinigung (an KS2)
      ;FOLD ;%{H}
         Case 141
      ;ENDFOLD
      ;FOLD -- RSK gestartet -- ;%{SE}%MKUKATPVW %CVW_COM %VCOMMENT %P 2:-- RSK gestartet --, 3: VW_COMMENT
      ;ENDFOLD
      ;FOLD F321 = AUS ;%{SE}%MKUKATPVW %CVW_SPS %VBOASG %P 2:F321 = AUS, 3: BOASG
         $FLAG[321] = FALSE
      ;ENDFOLD
      ;FOLD F323 = AUS ;%{SE}%MKUKATPVW %CVW_SPS %VBOASG %P 2:F323 = AUS, 3: BOASG
         $FLAG[323] = FALSE
      ;ENDFOLD
      ;FOLD F324 = AUS ;%{SE}%MKUKATPVW %CVW_SPS %VBOASG %P 2:F324 = AUS, 3: BOASG
         $FLAG[324] = FALSE
      ;ENDFOLD
      ;FOLD F329 = AUS ;%{SE}%MKUKATPVW %CVW_SPS %VBOASG %P 2:F329 = AUS, 3: BOASG
         $FLAG[329] = FALSE
      ;ENDFOLD
      ;FOLD -- MS2 Reinigung gestartet -- ;%{SE}%MKUKATPVW %CVW_COM %VCOMMENT %P 2:-- MS2 Reinigung gestartet --, 3: VW_COMMENT
      ;ENDFOLD
      ;FOLD F608 = EIN ;%{SE}%MKUKATPVW %CVW_SPS %VBOASG %P 2:F608 = EIN, 3: BOASG
         $FLAG[608] = TRUE
      ;ENDFOLD
      ;FOLD -- Ueberwachungszeit KS2 schwenken -- ;%{SE}%MKUKATPVW %CVW_COM %VCOMMENT %P 2:-- Ueberwachungszeit KS2 schwenken --, 3: VW_COMMENT
      ;ENDFOLD
      ;FOLD t8 ( EIN ) = -50[1/10Sek] ;%{SE}%MKUKATPVW %CVW_SPS %VTASG %P 2:t8 ( EIN ) = -50[1/10Sek], 3: TASG
         VW(#SET_TIME,TRUE,8,0,-50)
      ;ENDFOLD
      ;FOLD Schritt 142 = A4039 ;%{SE}%MKUKATPVW %CVW_SPS %VST_CON %P 2:Schritt 142 = A4039, 3: ST_CON
         IF $OUT[4039] THEN
            PREVSTEP = $APP_INT[5]
            $APP_INT[5] = 142
         ENDIF
      ;ENDFOLD
   ;ENDFOLD
   ;FOLD SCHRITT 142 -- MS2 Reinigung (an KS2) -- ;%{P}%MKUKATPVW,%CSTEP,%VST_NR,%P 1:SCHRITT, 2:142, 3: MS2 Reinigung (an KS2)
      ;FOLD ;%{H}
         Case 142
      ;ENDFOLD
      ;FOLD -- RSK Fehlerausgabe KS2 Ruhest. -- ;%{SE}%MKUKATPVW %CVW_COM %VCOMMENT %P 2:-- RSK Fehlerausgabe KS2 Ruhest. --, 3: VW_COMMENT
      ;ENDFOLD
      ;FOLD F323 = !E996 ;%{SE}%MKUKATPVW %CVW_SPS %VBOASG %P 2:F323 = !E996, 3: BOASG
         $FLAG[323] = NOT $IN[996]
      ;ENDFOLD
      ;FOLD -- RSK Sammelstoerung -- ;%{SE}%MKUKATPVW %CVW_COM %VCOMMENT %P 2:-- RSK Sammelstoerung --, 3: VW_COMMENT
      ;ENDFOLD
      ;FOLD F329 = F323 ;%{SE}%MKUKATPVW %CVW_SPS %VBOASG %P 2:F329 = F323, 3: BOASG
         $FLAG[329] = $FLAG[323]
      ;ENDFOLD
      ;FOLD Schritt 141 = (E26 + E27) & F323 & A4039 ;%{SE}%MKUKATPVW %CVW_SPS %VST_CON %P 2:Schritt 141 = (E26 + E27) & F323 & A4039, 3: ST_CON
         IF ($IN[26] OR $IN[27]) AND $FLAG[323] AND $OUT[4039] THEN
            PREVSTEP = $APP_INT[5]
            $APP_INT[5] = 141
         ENDIF
      ;ENDFOLD
      ;FOLD Schritt 143 = (!F323 + T8) & A4039 ;%{SE}%MKUKATPVW %CVW_SPS %VST_CON %P 2:Schritt 143 = (!F323 + T8) & A4039, 3: ST_CON
         IF (NOT $FLAG[323] OR $TIMER_FLAG[8]) AND $OUT[4039] THEN
            PREVSTEP = $APP_INT[5]
            $APP_INT[5] = 143
         ENDIF
      ;ENDFOLD
   ;ENDFOLD
   ;FOLD SCHRITT 143 -- MS2 Reinigung (an KS2) -- ;%{P}%MKUKATPVW,%CSTEP,%VST_NR,%P 1:SCHRITT, 2:143, 3: MS2 Reinigung (an KS2)
      ;FOLD ;%{H}
         Case 143
      ;ENDFOLD
      ;FOLD -- KS2 in Arbeitsstellung schwenken -- ;%{SE}%MKUKATPVW %CVW_COM %VCOMMENT %P 2:-- KS2 in Arbeitsstellung schwenken --, 3: VW_COMMENT
      ;ENDFOLD
      ;FOLD A1000 = !E997 ;%{SE}%MKUKATPVW %CVW_SPS %VBOASG %P 2:A1000 = !E997, 3: BOASG
         $OUT[1000] = NOT $IN[997]
      ;ENDFOLD
      ;FOLD Schritt 144 = A4039 ;%{SE}%MKUKATPVW %CVW_SPS %VST_CON %P 2:Schritt 144 = A4039, 3: ST_CON
         IF $OUT[4039] THEN
            PREVSTEP = $APP_INT[5]
            $APP_INT[5] = 144
         ENDIF
      ;ENDFOLD
   ;ENDFOLD
   ;FOLD SCHRITT 144 -- MS2 Reinigung (an KS2) -- ;%{P}%MKUKATPVW,%CSTEP,%VST_NR,%P 1:SCHRITT, 2:144, 3: MS2 Reinigung (an KS2)
      ;FOLD ;%{H}
         Case 144
      ;ENDFOLD
      ;FOLD -- RSK Fehlerausgabe KS2 Arbeitsstellung -- ;%{SE}%MKUKATPVW %CVW_COM %VCOMMENT %P 2:-- RSK Fehlerausgabe KS2 Arbeitsstellung --, 3: VW_COMMENT
      ;ENDFOLD
      ;FOLD F324 = !E997 & T8 + F324 ;%{SE}%MKUKATPVW %CVW_SPS %VBOASG %P 2:F324 = !E997 & T8 + F324, 3: BOASG
         $FLAG[324] = NOT $IN[997] AND $TIMER_FLAG[8] OR $FLAG[324]
      ;ENDFOLD
      ;FOLD -- RSK Sammelstoerung -- ;%{SE}%MKUKATPVW %CVW_COM %VCOMMENT %P 2:-- RSK Sammelstoerung --, 3: VW_COMMENT
      ;ENDFOLD
      ;FOLD F329 = F324 ;%{SE}%MKUKATPVW %CVW_SPS %VBOASG %P 2:F329 = F324, 3: BOASG
         $FLAG[329] = $FLAG[324]
      ;ENDFOLD
      ;FOLD Schritt 141 = F324 & (E26 + E27) & A4039 ;%{SE}%MKUKATPVW %CVW_SPS %VST_CON %P 2:Schritt 141 = F324 & (E26 + E27) & A4039, 3: ST_CON
         IF $FLAG[324] AND ($IN[26] OR $IN[27]) AND $OUT[4039] THEN
            PREVSTEP = $APP_INT[5]
            $APP_INT[5] = 141
         ENDIF
      ;ENDFOLD
      ;FOLD Schritt 145 = !F324 & E997 & !E999 & A4039 ;%{SE}%MKUKATPVW %CVW_SPS %VST_CON %P 2:Schritt 145 = !F324 & E997 & !E999 & A4039, 3: ST_CON
         IF NOT $FLAG[324] AND $IN[997] AND NOT $IN[999] AND $OUT[4039] THEN
            PREVSTEP = $APP_INT[5]
            $APP_INT[5] = 145
         ENDIF
      ;ENDFOLD
   ;ENDFOLD
   ;FOLD SCHRITT 145 -- MS2 Reinigung (an KS2) -- ;%{P}%MKUKATPVW,%CSTEP,%VST_NR,%P 1:SCHRITT, 2:145, 3: MS2 Reinigung (an KS2)
      ;FOLD ;%{H}
         Case 145
      ;ENDFOLD
      ;FOLD A1896 = AUS ;%{SE}%MKUKATPVW %CVW_SPS %VBOASG %P 2:A1896 = AUS, 3: BOASG
         $OUT[1896] = FALSE
      ;ENDFOLD
      ;FOLD A2176 = AUS ;%{SE}%MKUKATPVW %CVW_SPS %VBOASG %P 2:A2176 = AUS, 3: BOASG
         $OUT[2176] = FALSE
      ;ENDFOLD
      ;FOLD -- Ueberwachungszeit Versetzeinheit -- ;%{SE}%MKUKATPVW %CVW_COM %VCOMMENT %P 2:-- Ueberwachungszeit Versetzeinheit --, 3: VW_COMMENT
      ;ENDFOLD
      ;FOLD t8 ( EIN ) = -50[1/10Sek] ;%{SE}%MKUKATPVW %CVW_SPS %VTASG %P 2:t8 ( EIN ) = -50[1/10Sek], 3: TASG
         VW(#SET_TIME,TRUE,8,0,-50)
      ;ENDFOLD
      ;FOLD -- Ueberwachungszeit Reinigung -- ;%{SE}%MKUKATPVW %CVW_COM %VCOMMENT %P 2:-- Ueberwachungszeit Reinigung --, 3: VW_COMMENT
      ;ENDFOLD
      ;FOLD t9 ( EIN ) = -80[1/10Sek] ;%{SE}%MKUKATPVW %CVW_SPS %VTASG %P 2:t9 ( EIN ) = -80[1/10Sek], 3: TASG
         VW(#SET_TIME,TRUE,9,0,-80)
      ;ENDFOLD
      ;FOLD Schritt 146 = A4039 ;%{SE}%MKUKATPVW %CVW_SPS %VST_CON %P 2:Schritt 146 = A4039, 3: ST_CON
         IF $OUT[4039] THEN
            PREVSTEP = $APP_INT[5]
            $APP_INT[5] = 146
         ENDIF
      ;ENDFOLD
   ;ENDFOLD
   ;FOLD SCHRITT 146 -- MS2 Reinigung (an KS2) -- ;%{P}%MKUKATPVW,%CSTEP,%VST_NR,%P 1:SCHRITT, 2:146, 3: MS2 Reinigung (an KS2)
      ;FOLD ;%{H}
         Case 146
      ;ENDFOLD
      ;FOLD -- RSK Fehlerausgabe Versetzeinheit -- ;%{SE}%MKUKATPVW %CVW_COM %VCOMMENT %P 2:-- RSK Fehlerausgabe Versetzeinheit --, 3: VW_COMMENT
      ;ENDFOLD
      ;FOLD F328 = F585 & T8 ;%{SE}%MKUKATPVW %CVW_SPS %VBOASG %P 2:F328 = F585 & T8, 3: BOASG
         $FLAG[328] = $FLAG[585] AND $TIMER_FLAG[8]
      ;ENDFOLD
      ;FOLD -- RSK Sammelstoerung -- ;%{SE}%MKUKATPVW %CVW_COM %VCOMMENT %P 2:-- RSK Sammelstoerung --, 3: VW_COMMENT
      ;ENDFOLD
      ;FOLD F329 = T8 ;%{SE}%MKUKATPVW %CVW_SPS %VBOASG %P 2:F329 = T8, 3: BOASG
         $FLAG[329] = $TIMER_FLAG[8]
      ;ENDFOLD
      ;FOLD -- Versetzeinheit in Arbeitsst. schw. -- ;%{SE}%MKUKATPVW %CVW_COM %VCOMMENT %P 2:-- Versetzeinheit in Arbeitsst. schw. --, 3: VW_COMMENT
      ;ENDFOLD
      ;FOLD A2176 = !E2176 & F585 ;%{SE}%MKUKATPVW %CVW_SPS %VBOASG %P 2:A2176 = !E2176 & F585, 3: BOASG
         $OUT[2176] = NOT $IN[2176] AND $FLAG[585]
      ;ENDFOLD
      ;FOLD Schritt 145 = A2176 & T8 & (E26 + E27) & A4039 ;%{SE}%MKUKATPVW %CVW_SPS %VST_CON %P 2:Schritt 145 = A2176 & T8 & (E26 + E27) & A4039, 3: ST_CON
         IF $OUT[2176] AND $TIMER_FLAG[8] AND ($IN[26] OR $IN[27]) AND $OUT[4039] THEN
            PREVSTEP = $APP_INT[5]
            $APP_INT[5] = 145
         ENDIF
      ;ENDFOLD
      ;FOLD Schritt 147 = (E2176 & F585 + !E2168 & !F585) & A4039 ;%{SE}%MKUKATPVW %CVW_SPS %VST_CON %P 2:Schritt 147 = (E2176 & F585 + !E2168 & !F585) & A4039, 3: ST_CON
         IF ($IN[2176] AND $FLAG[585] OR NOT $IN[2168] AND NOT $FLAG[585]) AND $OUT[4039] THEN
            PREVSTEP = $APP_INT[5]
            $APP_INT[5] = 147
         ENDIF
      ;ENDFOLD
   ;ENDFOLD
   ;FOLD SCHRITT 147 -- MS2 Reinigung (an KS2) -- ;%{P}%MKUKATPVW,%CSTEP,%VST_NR,%P 1:SCHRITT, 2:147, 3: MS2 Reinigung (an KS2)
      ;FOLD ;%{H}
         Case 147
      ;ENDFOLD
      ;FOLD -- RSK Sammelstoerung -- ;%{SE}%MKUKATPVW %CVW_COM %VCOMMENT %P 2:-- RSK Sammelstoerung --, 3: VW_COMMENT
      ;ENDFOLD
      ;FOLD F329 = T9 ;%{SE}%MKUKATPVW %CVW_SPS %VBOASG %P 2:F329 = T9, 3: BOASG
         $FLAG[329] = $TIMER_FLAG[9]
      ;ENDFOLD
      ;FOLD -- MS2 Ausblasen EIN -- ;%{SE}%MKUKATPVW %CVW_COM %VCOMMENT %P 2:-- MS2 Ausblasen EIN --, 3: VW_COMMENT
      ;ENDFOLD
      ;FOLD A1902 = EIN ;%{SE}%MKUKATPVW %CVW_SPS %VBOASG %P 2:A1902 = EIN, 3: BOASG
         $OUT[1902] = TRUE
      ;ENDFOLD
      ;FOLD -- MS2 Reinigung starten -- ;%{SE}%MKUKATPVW %CVW_COM %VCOMMENT %P 2:-- MS2 Reinigung starten --, 3: VW_COMMENT
      ;ENDFOLD
      ;FOLD A1896 = EIN ;%{SE}%MKUKATPVW %CVW_SPS %VBOASG %P 2:A1896 = EIN, 3: BOASG
         $OUT[1896] = TRUE
      ;ENDFOLD
      ;FOLD Schritt 145 = !E1896 & T9 & (E26 + E27) & A4039 ;%{SE}%MKUKATPVW %CVW_SPS %VST_CON %P 2:Schritt 145 = !E1896 & T9 & (E26 + E27) & A4039, 3: ST_CON
         IF NOT $IN[1896] AND $TIMER_FLAG[9] AND ($IN[26] OR $IN[27]) AND $OUT[4039] THEN
            PREVSTEP = $APP_INT[5]
            $APP_INT[5] = 145
         ENDIF
      ;ENDFOLD
      ;FOLD Schritt 148 = E1896 & A4039 ;%{SE}%MKUKATPVW %CVW_SPS %VST_CON %P 2:Schritt 148 = E1896 & A4039, 3: ST_CON
         IF $IN[1896] AND $OUT[4039] THEN
            PREVSTEP = $APP_INT[5]
            $APP_INT[5] = 148
         ENDIF
      ;ENDFOLD
   ;ENDFOLD
   ;FOLD SCHRITT 148 -- MS2 Reinigung (an KS2) -- ;%{P}%MKUKATPVW,%CSTEP,%VST_NR,%P 1:SCHRITT, 2:148, 3: MS2 Reinigung (an KS2)
      ;FOLD ;%{H}
         Case 148
      ;ENDFOLD
      ;FOLD -- MS2 Reinigung beenden -- ;%{SE}%MKUKATPVW %CVW_COM %VCOMMENT %P 2:-- MS2 Reinigung beenden --, 3: VW_COMMENT
      ;ENDFOLD
      ;FOLD A1896 = AUS ;%{SE}%MKUKATPVW %CVW_SPS %VBOASG %P 2:A1896 = AUS, 3: BOASG
         $OUT[1896] = FALSE
      ;ENDFOLD
      ;FOLD -- MS2 Ausblasen AUS -- ;%{SE}%MKUKATPVW %CVW_COM %VCOMMENT %P 2:-- MS2 Ausblasen AUS --, 3: VW_COMMENT
      ;ENDFOLD
      ;FOLD A1902 = AUS ;%{SE}%MKUKATPVW %CVW_SPS %VBOASG %P 2:A1902 = AUS, 3: BOASG
         $OUT[1902] = FALSE
      ;ENDFOLD
      ;FOLD -- MS2 Einspruehen EIN -- ;%{SE}%MKUKATPVW %CVW_COM %VCOMMENT %P 2:-- MS2 Einspruehen EIN --, 3: VW_COMMENT
      ;ENDFOLD
      ;FOLD A528 = !F583 & F584 ;%{SE}%MKUKATPVW %CVW_SPS %VBOASG %P 2:A528 = !F583 & F584, 3: BOASG
         $OUT[528] = NOT $FLAG[583] AND $FLAG[584]
      ;ENDFOLD
      ;FOLD A1903 = F583 & F584 ;%{SE}%MKUKATPVW %CVW_SPS %VBOASG %P 2:A1903 = F583 & F584, 3: BOASG
         $OUT[1903] = $FLAG[583] AND $FLAG[584]
      ;ENDFOLD
      ;FOLD -- Einschaltdauer Einspruehen -- ;%{SE}%MKUKATPVW %CVW_COM %VCOMMENT %P 2:-- Einschaltdauer Einspruehen --, 3: VW_COMMENT
      ;ENDFOLD
      ;FOLD t7 ( EIN ) = i23[1/10Sek] ;%{SE}%MKUKATPVW %CVW_SPS %VTASG %P 2:t7 ( EIN ) = i23[1/10Sek], 3: TASG
         VW(#SET_TIME,TRUE,7,0,$COUNT_I[23])
      ;ENDFOLD
      ;FOLD Schritt 149 = A4039 ;%{SE}%MKUKATPVW %CVW_SPS %VST_CON %P 2:Schritt 149 = A4039, 3: ST_CON
         IF $OUT[4039] THEN
            PREVSTEP = $APP_INT[5]
            $APP_INT[5] = 149
         ENDIF
      ;ENDFOLD
   ;ENDFOLD
   ;FOLD SCHRITT 149 -- MS2 Reinigung (an KS2) -- ;%{P}%MKUKATPVW,%CSTEP,%VST_NR,%P 1:SCHRITT, 2:149, 3: MS2 Reinigung (an KS2)
      ;FOLD ;%{H}
         Case 149
      ;ENDFOLD
      ;FOLD F323 = AUS ;%{SE}%MKUKATPVW %CVW_SPS %VBOASG %P 2:F323 = AUS, 3: BOASG
         $FLAG[323] = FALSE
      ;ENDFOLD
      ;FOLD -- Ueberwachungszeit KS2 schwenken -- ;%{SE}%MKUKATPVW %CVW_COM %VCOMMENT %P 2:-- Ueberwachungszeit KS2 schwenken --, 3: VW_COMMENT
      ;ENDFOLD
      ;FOLD t8 ( EIN ) = -100[1/10Sek] ;%{SE}%MKUKATPVW %CVW_SPS %VTASG %P 2:t8 ( EIN ) = -100[1/10Sek], 3: TASG
         VW(#SET_TIME,TRUE,8,0,-100)
      ;ENDFOLD
      ;FOLD Schritt 150 = T7 & A4039 ;%{SE}%MKUKATPVW %CVW_SPS %VST_CON %P 2:Schritt 150 = T7 & A4039, 3: ST_CON
         IF $TIMER_FLAG[7] AND $OUT[4039] THEN
            PREVSTEP = $APP_INT[5]
            $APP_INT[5] = 150
         ENDIF
      ;ENDFOLD
   ;ENDFOLD
   ;FOLD SCHRITT 150 -- MS2 Reinigung (an KS2) -- ;%{P}%MKUKATPVW,%CSTEP,%VST_NR,%P 1:SCHRITT, 2:150, 3: MS2 Reinigung (an KS2)
      ;FOLD ;%{H}
         Case 150
      ;ENDFOLD
      ;FOLD -- MS2 Einspruehen AUS -- ;%{SE}%MKUKATPVW %CVW_COM %VCOMMENT %P 2:-- MS2 Einspruehen AUS --, 3: VW_COMMENT
      ;ENDFOLD
      ;FOLD A528 = AUS ;%{SE}%MKUKATPVW %CVW_SPS %VBOASG %P 2:A528 = AUS, 3: BOASG
         $OUT[528] = FALSE
      ;ENDFOLD
      ;FOLD A1903 = AUS ;%{SE}%MKUKATPVW %CVW_SPS %VBOASG %P 2:A1903 = AUS, 3: BOASG
         $OUT[1903] = FALSE
      ;ENDFOLD
      ;FOLD -- RSK Fehlerausgabe KS2 Ruhest. -- ;%{SE}%MKUKATPVW %CVW_COM %VCOMMENT %P 2:-- RSK Fehlerausgabe KS2 Ruhest. --, 3: VW_COMMENT
      ;ENDFOLD
      ;FOLD F324 = !E997 ;%{SE}%MKUKATPVW %CVW_SPS %VBOASG %P 2:F324 = !E997, 3: BOASG
         $FLAG[324] = NOT $IN[997]
      ;ENDFOLD
      ;FOLD -- RSK Sammelstoerung -- ;%{SE}%MKUKATPVW %CVW_COM %VCOMMENT %P 2:-- RSK Sammelstoerung --, 3: VW_COMMENT
      ;ENDFOLD
      ;FOLD F329 = F324 ;%{SE}%MKUKATPVW %CVW_SPS %VBOASG %P 2:F329 = F324, 3: BOASG
         $FLAG[329] = $FLAG[324]
      ;ENDFOLD
      ;FOLD Schritt 149 = (E26 + E27) & F324 & A4039 ;%{SE}%MKUKATPVW %CVW_SPS %VST_CON %P 2:Schritt 149 = (E26 + E27) & F324 & A4039, 3: ST_CON
         IF ($IN[26] OR $IN[27]) AND $FLAG[324] AND $OUT[4039] THEN
            PREVSTEP = $APP_INT[5]
            $APP_INT[5] = 149
         ENDIF
      ;ENDFOLD
      ;FOLD Schritt 151 = (!F324 + T8) & A4039 ;%{SE}%MKUKATPVW %CVW_SPS %VST_CON %P 2:Schritt 151 = (!F324 + T8) & A4039, 3: ST_CON
         IF (NOT $FLAG[324] OR $TIMER_FLAG[8]) AND $OUT[4039] THEN
            PREVSTEP = $APP_INT[5]
            $APP_INT[5] = 151
         ENDIF
      ;ENDFOLD
   ;ENDFOLD
   ;FOLD SCHRITT 151 -- MS2 Reinigung (an KS2) -- ;%{P}%MKUKATPVW,%CSTEP,%VST_NR,%P 1:SCHRITT, 2:151, 3: MS2 Reinigung (an KS2)
      ;FOLD ;%{H}
         Case 151
      ;ENDFOLD
      ;FOLD -- KS2 in Ruhestellung schwenken -- ;%{SE}%MKUKATPVW %CVW_COM %VCOMMENT %P 2:-- KS2 in Ruhestellung schwenken --, 3: VW_COMMENT
      ;ENDFOLD
      ;FOLD A1000 = !E996 ;%{SE}%MKUKATPVW %CVW_SPS %VBOASG %P 2:A1000 = !E996, 3: BOASG
         $OUT[1000] = NOT $IN[996]
      ;ENDFOLD
      ;FOLD Schritt 152 = A4039 ;%{SE}%MKUKATPVW %CVW_SPS %VST_CON %P 2:Schritt 152 = A4039, 3: ST_CON
         IF $OUT[4039] THEN
            PREVSTEP = $APP_INT[5]
            $APP_INT[5] = 152
         ENDIF
      ;ENDFOLD
   ;ENDFOLD
   ;FOLD SCHRITT 152 -- MS2 Reinigung (an KS2) -- ;%{P}%MKUKATPVW,%CSTEP,%VST_NR,%P 1:SCHRITT, 2:152, 3: MS2 Reinigung (an KS2)
      ;FOLD ;%{H}
         Case 152
      ;ENDFOLD
      ;FOLD -- RSK Fehlerausgabe KS2 Ruhestellung -- ;%{SE}%MKUKATPVW %CVW_COM %VCOMMENT %P 2:-- RSK Fehlerausgabe KS2 Ruhestellung --, 3: VW_COMMENT
      ;ENDFOLD
      ;FOLD F323 = !E996 & T8 + F323 ;%{SE}%MKUKATPVW %CVW_SPS %VBOASG %P 2:F323 = !E996 & T8 + F323, 3: BOASG
         $FLAG[323] = NOT $IN[996] AND $TIMER_FLAG[8] OR $FLAG[323]
      ;ENDFOLD
      ;FOLD -- RSK Sammelstoerung -- ;%{SE}%MKUKATPVW %CVW_COM %VCOMMENT %P 2:-- RSK Sammelstoerung --, 3: VW_COMMENT
      ;ENDFOLD
      ;FOLD F329 = F323 ;%{SE}%MKUKATPVW %CVW_SPS %VBOASG %P 2:F329 = F323, 3: BOASG
         $FLAG[329] = $FLAG[323]
      ;ENDFOLD
      ;FOLD Schritt 149 = F323 & (E26 + E27) & A4039 ;%{SE}%MKUKATPVW %CVW_SPS %VST_CON %P 2:Schritt 149 = F323 & (E26 + E27) & A4039, 3: ST_CON
         IF $FLAG[323] AND ($IN[26] OR $IN[27]) AND $OUT[4039] THEN
            PREVSTEP = $APP_INT[5]
            $APP_INT[5] = 149
         ENDIF
      ;ENDFOLD
      ;FOLD Schritt 153 = E996 & !E998 & A4039 ;%{SE}%MKUKATPVW %CVW_SPS %VST_CON %P 2:Schritt 153 = E996 & !E998 & A4039, 3: ST_CON
         IF $IN[996] AND NOT $IN[998] AND $OUT[4039] THEN
            PREVSTEP = $APP_INT[5]
            $APP_INT[5] = 153
         ENDIF
      ;ENDFOLD
   ;ENDFOLD
   ;FOLD SCHRITT 153 -- MS2 Reinigung (an KS2) -- ;%{P}%MKUKATPVW,%CSTEP,%VST_NR,%P 1:SCHRITT, 2:153, 3: MS2 Reinigung (an KS2)
      ;FOLD ;%{H}
         Case 153
      ;ENDFOLD
      ;FOLD F323 = AUS ;%{SE}%MKUKATPVW %CVW_SPS %VBOASG %P 2:F323 = AUS, 3: BOASG
         $FLAG[323] = FALSE
      ;ENDFOLD
      ;FOLD F329 = AUS ;%{SE}%MKUKATPVW %CVW_SPS %VBOASG %P 2:F329 = AUS, 3: BOASG
         $FLAG[329] = FALSE
      ;ENDFOLD
      ;FOLD -- MS2 Zaehler ruecksetzen -- ;%{SE}%MKUKATPVW %CVW_COM %VCOMMENT %P 2:-- MS2 Zaehler ruecksetzen --, 3: VW_COMMENT
      ;ENDFOLD
      ;FOLD -- MS2 FRG Reinigung -- ;%{SE}%MKUKATPVW %CVW_COM %VCOMMENT %P 2:-- MS2 FRG Reinigung --, 3: VW_COMMENT
      ;ENDFOLD
      ;FOLD F607 = AUS ;%{SE}%MKUKATPVW %CVW_SPS %VBOASG %P 2:F607 = AUS, 3: BOASG
         $FLAG[607] = FALSE
      ;ENDFOLD
      ;FOLD -- MS2 Reinigung FK -- ;%{SE}%MKUKATPVW %CVW_COM %VCOMMENT %P 2:-- MS2 Reinigung FK --, 3: VW_COMMENT
      ;ENDFOLD
      ;FOLD F609 = EIN ;%{SE}%MKUKATPVW %CVW_SPS %VBOASG %P 2:F609 = EIN, 3: BOASG
         $FLAG[609] = TRUE
      ;ENDFOLD
      ;FOLD t8 ( EIN ) = STOP ;%{SE}%MKUKATPVW %CVW_SPS %VTSTOP %P 2:t8 ( EIN ) = STOP, 3: TSTOP
         VW(#SET_TIME,TRUE,8,1,0)
      ;ENDFOLD
      ;FOLD Schritt 1 = A4039 ;%{SE}%MKUKATPVW %CVW_SPS %VST_CON %P 2:Schritt 1 = A4039, 3: ST_CON
         IF $OUT[4039] THEN
            PREVSTEP = $APP_INT[5]
            $APP_INT[5] = 1
         ENDIF
      ;ENDFOLD
   ;ENDFOLD
   ;FOLD SCHRITT 154 -- MS1 Reinigung (an Pneum. Schwenkeinheit MS1)-- ;%{P}%MKUKATPVW,%CSTEP,%VST_NR,%P 1:SCHRITT, 2:154, 3: MS1 Reinigung (an Pneum. Schwenkeinheit MS1)
      ;FOLD ;%{H}
         Case 154
      ;ENDFOLD
      ;FOLD -- RSK gestartet -- ;%{SE}%MKUKATPVW %CVW_COM %VCOMMENT %P 2:-- RSK gestartet --, 3: VW_COMMENT
      ;ENDFOLD
      ;FOLD F321 = AUS ;%{SE}%MKUKATPVW %CVW_SPS %VBOASG %P 2:F321 = AUS, 3: BOASG
         $FLAG[321] = FALSE
      ;ENDFOLD
      ;FOLD F323 = AUS ;%{SE}%MKUKATPVW %CVW_SPS %VBOASG %P 2:F323 = AUS, 3: BOASG
         $FLAG[323] = FALSE
      ;ENDFOLD
      ;FOLD F324 = AUS ;%{SE}%MKUKATPVW %CVW_SPS %VBOASG %P 2:F324 = AUS, 3: BOASG
         $FLAG[324] = FALSE
      ;ENDFOLD
      ;FOLD F329 = AUS ;%{SE}%MKUKATPVW %CVW_SPS %VBOASG %P 2:F329 = AUS, 3: BOASG
         $FLAG[329] = FALSE
      ;ENDFOLD
      ;FOLD -- MS1 Reinigung gestartet -- ;%{SE}%MKUKATPVW %CVW_COM %VCOMMENT %P 2:-- MS1 Reinigung gestartet --, 3: VW_COMMENT
      ;ENDFOLD
      ;FOLD F604 = EIN ;%{SE}%MKUKATPVW %CVW_SPS %VBOASG %P 2:F604 = EIN, 3: BOASG
         $FLAG[604] = TRUE
      ;ENDFOLD
      ;FOLD -- Steuerluft EIN -- ;%{SE}%MKUKATPVW %CVW_COM %VCOMMENT %P 2:-- Steuerluft EIN --, 3: VW_COMMENT
      ;ENDFOLD
      ;FOLD A2161 = A4039 ;%{SE}%MKUKATPVW %CVW_SPS %VBOASG %P 2:A2161 = A4039, 3: BOASG
         $OUT[2161] = $OUT[4039]
      ;ENDFOLD
      ;FOLD A2163 = AUS ;%{SE}%MKUKATPVW %CVW_SPS %VBOASG %P 2:A2163 = AUS, 3: BOASG
         $OUT[2163] = FALSE
      ;ENDFOLD
      ;FOLD A2164 = AUS ;%{SE}%MKUKATPVW %CVW_SPS %VBOASG %P 2:A2164 = AUS, 3: BOASG
         $OUT[2164] = FALSE
      ;ENDFOLD
      ;FOLD A2165 = AUS ;%{SE}%MKUKATPVW %CVW_SPS %VBOASG %P 2:A2165 = AUS, 3: BOASG
         $OUT[2165] = FALSE
      ;ENDFOLD
      ;FOLD A2166 = AUS ;%{SE}%MKUKATPVW %CVW_SPS %VBOASG %P 2:A2166 = AUS, 3: BOASG
         $OUT[2166] = FALSE
      ;ENDFOLD
      ;FOLD A2167 = AUS ;%{SE}%MKUKATPVW %CVW_SPS %VBOASG %P 2:A2167 = AUS, 3: BOASG
         $OUT[2167] = FALSE
      ;ENDFOLD
      ;FOLD A2168 = AUS ;%{SE}%MKUKATPVW %CVW_SPS %VBOASG %P 2:A2168 = AUS, 3: BOASG
         $OUT[2168] = FALSE
      ;ENDFOLD
      ;FOLD -- Ueberwachungszeit Schwenkeinheit 1 -- ;%{SE}%MKUKATPVW %CVW_COM %VCOMMENT %P 2:-- Ueberwachungszeit Schwenkeinheit 1 --, 3: VW_COMMENT
      ;ENDFOLD
      ;FOLD t8 ( EIN ) = -100[1/10Sek] ;%{SE}%MKUKATPVW %CVW_SPS %VTASG %P 2:t8 ( EIN ) = -100[1/10Sek], 3: TASG
         VW(#SET_TIME,TRUE,8,0,-100)
      ;ENDFOLD
      ;FOLD Schritt 155 = A4039 ;%{SE}%MKUKATPVW %CVW_SPS %VST_CON %P 2:Schritt 155 = A4039, 3: ST_CON
         IF $OUT[4039] THEN
            PREVSTEP = $APP_INT[5]
            $APP_INT[5] = 155
         ENDIF
      ;ENDFOLD
   ;ENDFOLD
   ;FOLD SCHRITT 155 -- MS1 Reinigung (an Pneum. Schwenkeinheit MS1)-- ;%{P}%MKUKATPVW,%CSTEP,%VST_NR,%P 1:SCHRITT, 2:155, 3: MS1 Reinigung (an Pneum. Schwenkeinheit MS1)
      ;FOLD ;%{H}
         Case 155
      ;ENDFOLD
      ;FOLD -- Steuerluft EIN -- ;%{SE}%MKUKATPVW %CVW_COM %VCOMMENT %P 2:-- Steuerluft EIN --, 3: VW_COMMENT
      ;ENDFOLD
      ;FOLD A2161 = A4039 ;%{SE}%MKUKATPVW %CVW_SPS %VBOASG %P 2:A2161 = A4039, 3: BOASG
         $OUT[2161] = $OUT[4039]
      ;ENDFOLD
      ;FOLD -- RSK Fehlerausgabe Schwenkeinheit 1 Ruhest. -- ;%{SE}%MKUKATPVW %CVW_COM %VCOMMENT %P 2:-- RSK Fehlerausgabe Schwenkeinheit 1 Ruhest. --, 3: VW_COMMENT
      ;ENDFOLD
      ;FOLD F323 = !E2163 & T8 ;%{SE}%MKUKATPVW %CVW_SPS %VBOASG %P 2:F323 = !E2163 & T8, 3: BOASG
         $FLAG[323] = NOT $IN[2163] AND $TIMER_FLAG[8]
      ;ENDFOLD
      ;FOLD -- RSK Sammelstoerung -- ;%{SE}%MKUKATPVW %CVW_COM %VCOMMENT %P 2:-- RSK Sammelstoerung --, 3: VW_COMMENT
      ;ENDFOLD
      ;FOLD F329 = F323 + T8 ;%{SE}%MKUKATPVW %CVW_SPS %VBOASG %P 2:F329 = F323 + T8, 3: BOASG
         $FLAG[329] = $FLAG[323] OR $TIMER_FLAG[8]
      ;ENDFOLD
      ;FOLD Schritt 154 = (E26 + E27) & F323 & A4039 ;%{SE}%MKUKATPVW %CVW_SPS %VST_CON %P 2:Schritt 154 = (E26 + E27) & F323 & A4039, 3: ST_CON
         IF ($IN[26] OR $IN[27]) AND $FLAG[323] AND $OUT[4039] THEN
            PREVSTEP = $APP_INT[5]
            $APP_INT[5] = 154
         ENDIF
      ;ENDFOLD
      ;FOLD Schritt 156 = (!F323 + T8) & (F523 & !F524 & E2161 + !F523 & F524 & !E2162) & A4039 ;%{SE}%MKUKATPVW %CVW_SPS %VST_CON %P 2:Schritt 156 = (!F323 + T8) & (F523 & !F524 & E2161 + !F523 & F524 & !E2162) & A4039, 3: ST_CON
         IF (NOT $FLAG[323] OR $TIMER_FLAG[8]) AND ($FLAG[523] AND NOT $FLAG[524] AND $IN[2161] OR NOT $FLAG[523] AND $FLAG[524] AND NOT $IN[2162]) AND $OUT[4039] THEN
            PREVSTEP = $APP_INT[5]
            $APP_INT[5] = 156
         ENDIF
      ;ENDFOLD
   ;ENDFOLD
   ;FOLD SCHRITT 156 -- MS1 Reinigung (an Pneum. Schwenkeinheit MS1)-- ;%{P}%MKUKATPVW,%CSTEP,%VST_NR,%P 1:SCHRITT, 2:156, 3: MS1 Reinigung (an Pneum. Schwenkeinheit MS1)
      ;FOLD ;%{H}
         Case 156
      ;ENDFOLD
      ;FOLD -- Steuerluft EIN -- ;%{SE}%MKUKATPVW %CVW_COM %VCOMMENT %P 2:-- Steuerluft EIN --, 3: VW_COMMENT
      ;ENDFOLD
      ;FOLD A2161 = A4039 ;%{SE}%MKUKATPVW %CVW_SPS %VBOASG %P 2:A2161 = A4039, 3: BOASG
         $OUT[2161] = $OUT[4039]
      ;ENDFOLD
      ;FOLD -- Schwenkeinheit 1 in Arbeitsstellung schwenken -- ;%{SE}%MKUKATPVW %CVW_COM %VCOMMENT %P 2:-- Schwenkeinheit 1 in Arbeitsstellung schwenken --, 3: VW_COMMENT
      ;ENDFOLD
      ;FOLD A2163 = AUS ;%{SE}%MKUKATPVW %CVW_SPS %VBOASG %P 2:A2163 = AUS, 3: BOASG
         $OUT[2163] = FALSE
      ;ENDFOLD
      ;FOLD A2164 = EIN ;%{SE}%MKUKATPVW %CVW_SPS %VBOASG %P 2:A2164 = EIN, 3: BOASG
         $OUT[2164] = TRUE
      ;ENDFOLD
      ;FOLD -- FRG Bewegung EIN -- ;%{SE}%MKUKATPVW %CVW_COM %VCOMMENT %P 2:-- FRG Bewegung EIN --, 3: VW_COMMENT
      ;ENDFOLD
      ;FOLD A2165 = AUS ;%{SE}%MKUKATPVW %CVW_SPS %VBOASG %P 2:A2165 = AUS, 3: BOASG
         $OUT[2165] = FALSE
      ;ENDFOLD
      ;FOLD A2166 = EIN ;%{SE}%MKUKATPVW %CVW_SPS %VBOASG %P 2:A2166 = EIN, 3: BOASG
         $OUT[2166] = TRUE
      ;ENDFOLD
      ;FOLD -- Zeit Endlage entprellen -- ;%{SE}%MKUKATPVW %CVW_COM %VCOMMENT %P 2:-- Zeit Endlage entprellen --, 3: VW_COMMENT
      ;ENDFOLD
      ;FOLD t9 ( !E2164 ) = -10[1/10Sek] ;%{SE}%MKUKATPVW %CVW_SPS %VTASG %P 2:t9 ( !E2164 ) = -10[1/10Sek], 3: TASG
         VW(#SET_TIME,NOT $IN[2164],9,0,-10)
      ;ENDFOLD
      ;FOLD Schritt 157 = E2164 & !E2163 & A4039 & T9 + T8 ;%{SE}%MKUKATPVW %CVW_SPS %VST_CON %P 2:Schritt 157 = E2164 & !E2163 & A4039 & T9 + T8, 3: ST_CON
         IF $IN[2164] AND NOT $IN[2163] AND $OUT[4039] AND $TIMER_FLAG[9] OR $TIMER_FLAG[8] THEN
            PREVSTEP = $APP_INT[5]
            $APP_INT[5] = 157
         ENDIF
      ;ENDFOLD
   ;ENDFOLD
   ;FOLD SCHRITT 157 -- MS1 Reinigung (an Pneum. Schwenkeinheit MS1)-- ;%{P}%MKUKATPVW,%CSTEP,%VST_NR,%P 1:SCHRITT, 2:157, 3: MS1 Reinigung (an Pneum. Schwenkeinheit MS1)
      ;FOLD ;%{H}
         Case 157
      ;ENDFOLD
      ;FOLD -- Steuerluft EIN -- ;%{SE}%MKUKATPVW %CVW_COM %VCOMMENT %P 2:-- Steuerluft EIN --, 3: VW_COMMENT
      ;ENDFOLD
      ;FOLD A2161 = A4039 ;%{SE}%MKUKATPVW %CVW_SPS %VBOASG %P 2:A2161 = A4039, 3: BOASG
         $OUT[2161] = $OUT[4039]
      ;ENDFOLD
      ;FOLD -- RSK Fehlerausgabe Schwenkeinheit 1 Arbeitsstellung -- ;%{SE}%MKUKATPVW %CVW_COM %VCOMMENT %P 2:-- RSK Fehlerausgabe Schwenkeinheit 1 Arbeitsstellung --, 3: VW_COMMENT
      ;ENDFOLD
      ;FOLD F324 = !E2164 & T8 + F324 ;%{SE}%MKUKATPVW %CVW_SPS %VBOASG %P 2:F324 = !E2164 & T8 + F324, 3: BOASG
         $FLAG[324] = NOT $IN[2164] AND $TIMER_FLAG[8] OR $FLAG[324]
      ;ENDFOLD
      ;FOLD -- RSK Sammelstoerung -- ;%{SE}%MKUKATPVW %CVW_COM %VCOMMENT %P 2:-- RSK Sammelstoerung --, 3: VW_COMMENT
      ;ENDFOLD
      ;FOLD F329 = F324 ;%{SE}%MKUKATPVW %CVW_SPS %VBOASG %P 2:F329 = F324, 3: BOASG
         $FLAG[329] = $FLAG[324]
      ;ENDFOLD
      ;FOLD A2164 = AUS ;%{SE}%MKUKATPVW %CVW_SPS %VBOASG %P 2:A2164 = AUS, 3: BOASG
         $OUT[2164] = FALSE
      ;ENDFOLD
      ;FOLD -- FRG Bewegung AUS -- ;%{SE}%MKUKATPVW %CVW_COM %VCOMMENT %P 2:-- FRG Bewegung AUS --, 3: VW_COMMENT
      ;ENDFOLD
      ;FOLD A2166 = AUS ;%{SE}%MKUKATPVW %CVW_SPS %VBOASG %P 2:A2166 = AUS, 3: BOASG
         $OUT[2166] = FALSE
      ;ENDFOLD
      ;FOLD -- FRG in Endlage halten ein -- ;%{SE}%MKUKATPVW %CVW_COM %VCOMMENT %P 2:-- FRG in Endlage halten ein --, 3: VW_COMMENT
      ;ENDFOLD
      ;FOLD A2165 = EIN ;%{SE}%MKUKATPVW %CVW_SPS %VBOASG %P 2:A2165 = EIN, 3: BOASG
         $OUT[2165] = TRUE
      ;ENDFOLD
      ;FOLD Schritt 154 = F324 & (E26 + E27) & A4039 ;%{SE}%MKUKATPVW %CVW_SPS %VST_CON %P 2:Schritt 154 = F324 & (E26 + E27) & A4039, 3: ST_CON
         IF $FLAG[324] AND ($IN[26] OR $IN[27]) AND $OUT[4039] THEN
            PREVSTEP = $APP_INT[5]
            $APP_INT[5] = 154
         ENDIF
      ;ENDFOLD
      ;FOLD Schritt 158 = !F324 & E2164 & A4039 ;%{SE}%MKUKATPVW %CVW_SPS %VST_CON %P 2:Schritt 158 = !F324 & E2164 & A4039, 3: ST_CON
         IF NOT $FLAG[324] AND $IN[2164] AND $OUT[4039] THEN
            PREVSTEP = $APP_INT[5]
            $APP_INT[5] = 158
         ENDIF
      ;ENDFOLD
   ;ENDFOLD
   ;FOLD SCHRITT 158 -- MS1 Reinigung (an Pneum. Schwenkeinheit MS1)-- ;%{P}%MKUKATPVW,%CSTEP,%VST_NR,%P 1:SCHRITT, 2:158, 3: MS1 Reinigung (an Pneum. Schwenkeinheit MS1)
      ;FOLD ;%{H}
         Case 158
      ;ENDFOLD
      ;FOLD -- Steuerluft EIN -- ;%{SE}%MKUKATPVW %CVW_COM %VCOMMENT %P 2:-- Steuerluft EIN --, 3: VW_COMMENT
      ;ENDFOLD
      ;FOLD A2161 = A4039 ;%{SE}%MKUKATPVW %CVW_SPS %VBOASG %P 2:A2161 = A4039, 3: BOASG
         $OUT[2161] = $OUT[4039]
      ;ENDFOLD
      ;FOLD A1864 = AUS ;%{SE}%MKUKATPVW %CVW_SPS %VBOASG %P 2:A1864 = AUS, 3: BOASG
         $OUT[1864] = FALSE
      ;ENDFOLD
      ;FOLD A2168 = AUS ;%{SE}%MKUKATPVW %CVW_SPS %VBOASG %P 2:A2168 = AUS, 3: BOASG
         $OUT[2168] = FALSE
      ;ENDFOLD
      ;FOLD -- Ueberwachungszeit Versetzeinheit/Brennerreinigung -- ;%{SE}%MKUKATPVW %CVW_COM %VCOMMENT %P 2:-- Ueberwachungszeit Versetzeinheit/Brennerreinigung --, 3: VW_COMMENT
      ;ENDFOLD
      ;FOLD t8 ( EIN ) = -100[1/10Sek] ;%{SE}%MKUKATPVW %CVW_SPS %VTASG %P 2:t8 ( EIN ) = -100[1/10Sek], 3: TASG
         VW(#SET_TIME,TRUE,8,0,-100)
      ;ENDFOLD
      ;FOLD Schritt 159 = A4039 ;%{SE}%MKUKATPVW %CVW_SPS %VST_CON %P 2:Schritt 159 = A4039, 3: ST_CON
         IF $OUT[4039] THEN
            PREVSTEP = $APP_INT[5]
            $APP_INT[5] = 159
         ENDIF
      ;ENDFOLD
   ;ENDFOLD
   ;FOLD SCHRITT 159 -- MS1 Reinigung (an Pneum. Schwenkeinheit MS1)-- ;%{P}%MKUKATPVW,%CSTEP,%VST_NR,%P 1:SCHRITT, 2:159, 3: MS1 Reinigung (an Pneum. Schwenkeinheit MS1)
      ;FOLD ;%{H}
         Case 159
      ;ENDFOLD
      ;FOLD -- Steuerluft EIN -- ;%{SE}%MKUKATPVW %CVW_COM %VCOMMENT %P 2:-- Steuerluft EIN --, 3: VW_COMMENT
      ;ENDFOLD
      ;FOLD A2161 = A4039 ;%{SE}%MKUKATPVW %CVW_SPS %VBOASG %P 2:A2161 = A4039, 3: BOASG
         $OUT[2161] = $OUT[4039]
      ;ENDFOLD
      ;FOLD -- RSK Fehlerausgabe Versetzeinheit -- ;%{SE}%MKUKATPVW %CVW_COM %VCOMMENT %P 2:-- RSK Fehlerausgabe Versetzeinheit --, 3: VW_COMMENT
      ;ENDFOLD
      ;FOLD F328 = F576 & T8 ;%{SE}%MKUKATPVW %CVW_SPS %VBOASG %P 2:F328 = F576 & T8, 3: BOASG
         $FLAG[328] = $FLAG[576] AND $TIMER_FLAG[8]
      ;ENDFOLD
      ;FOLD -- RSK Sammelstoerung -- ;%{SE}%MKUKATPVW %CVW_COM %VCOMMENT %P 2:-- RSK Sammelstoerung --, 3: VW_COMMENT
      ;ENDFOLD
      ;FOLD F329 = T8 ;%{SE}%MKUKATPVW %CVW_SPS %VBOASG %P 2:F329 = T8, 3: BOASG
         $FLAG[329] = $TIMER_FLAG[8]
      ;ENDFOLD
      ;FOLD -- Versetzeinheit  in  Arbeitsst.  schw. -- ;%{SE}%MKUKATPVW %CVW_COM %VCOMMENT %P 2:-- Versetzeinheit  in  Arbeitsst.  schw. --, 3: VW_COMMENT
      ;ENDFOLD
      ;FOLD A2168 = !E2168 & E2164 & F576 ;%{SE}%MKUKATPVW %CVW_SPS %VBOASG %P 2:A2168 = !E2168 & E2164 & F576, 3: BOASG
         $OUT[2168] = NOT $IN[2168] AND $IN[2164] AND $FLAG[576]
      ;ENDFOLD
      ;FOLD Schritt 158 = A2168 & T8 & (E26 + E27) & A4039 ;%{SE}%MKUKATPVW %CVW_SPS %VST_CON %P 2:Schritt 158 = A2168 & T8 & (E26 + E27) & A4039, 3: ST_CON
         IF $OUT[2168] AND $TIMER_FLAG[8] AND ($IN[26] OR $IN[27]) AND $OUT[4039] THEN
            PREVSTEP = $APP_INT[5]
            $APP_INT[5] = 158
         ENDIF
      ;ENDFOLD
      ;FOLD Schritt 160 = (E2168 & F576 + !E2168 & !F576) & A4039 ;%{SE}%MKUKATPVW %CVW_SPS %VST_CON %P 2:Schritt 160 = (E2168 & F576 + !E2168 & !F576) & A4039, 3: ST_CON
         IF ($IN[2168] AND $FLAG[576] OR NOT $IN[2168] AND NOT $FLAG[576]) AND $OUT[4039] THEN
            PREVSTEP = $APP_INT[5]
            $APP_INT[5] = 160
         ENDIF
      ;ENDFOLD
   ;ENDFOLD
   ;FOLD SCHRITT 160 --MS1 Reinigung (an Pneum. Schwenkeinheit MS1)-- ;%{P}%MKUKATPVW,%CSTEP,%VST_NR,%P 1:SCHRITT, 2:160, 3:MS1 Reinigung (an Pneum. Schwenkeinheit MS1)
      ;FOLD ;%{H}
         Case 160
      ;ENDFOLD
      ;FOLD -- Steuerluft EIN -- ;%{SE}%MKUKATPVW %CVW_COM %VCOMMENT %P 2:-- Steuerluft EIN --, 3: VW_COMMENT
      ;ENDFOLD
      ;FOLD A2161 = A4039 ;%{SE}%MKUKATPVW %CVW_SPS %VBOASG %P 2:A2161 = A4039, 3: BOASG
         $OUT[2161] = $OUT[4039]
      ;ENDFOLD
      ;FOLD -- RSK Sammelstoerung -- ;%{SE}%MKUKATPVW %CVW_COM %VCOMMENT %P 2:-- RSK Sammelstoerung --, 3: VW_COMMENT
      ;ENDFOLD
      ;FOLD F329 = T8 ;%{SE}%MKUKATPVW %CVW_SPS %VBOASG %P 2:F329 = T8, 3: BOASG
         $FLAG[329] = $TIMER_FLAG[8]
      ;ENDFOLD
      ;FOLD -- Zeit Reinigung -- ;%{SE}%MKUKATPVW %CVW_COM %VCOMMENT %P 2:-- Zeit Reinigung --, 3: VW_COMMENT
      ;ENDFOLD
      ;FOLD t9 ( EIN ) = -20[1/10Sek] ;%{SE}%MKUKATPVW %CVW_SPS %VTASG %P 2:t9 ( EIN ) = -20[1/10Sek], 3: TASG
         VW(#SET_TIME,TRUE,9,0,-20)
      ;ENDFOLD
      ;FOLD -- MS1 Ausblasen EIN -- ;%{SE}%MKUKATPVW %CVW_COM %VCOMMENT %P 2:-- MS1 Ausblasen EIN --, 3: VW_COMMENT
      ;ENDFOLD
      ;FOLD A1870 = EIN ;%{SE}%MKUKATPVW %CVW_SPS %VBOASG %P 2:A1870 = EIN, 3: BOASG
         $OUT[1870] = TRUE
      ;ENDFOLD
      ;FOLD -- MS1 Reinigung starten -- ;%{SE}%MKUKATPVW %CVW_COM %VCOMMENT %P 2:-- MS1 Reinigung starten --, 3: VW_COMMENT
      ;ENDFOLD
      ;FOLD A1864 = EIN ;%{SE}%MKUKATPVW %CVW_SPS %VBOASG %P 2:A1864 = EIN, 3: BOASG
         $OUT[1864] = TRUE
      ;ENDFOLD
      ;FOLD Schritt 158 = E1864 & T8 & (E26 + E27) & A4039 ;%{SE}%MKUKATPVW %CVW_SPS %VST_CON %P 2:Schritt 158 = E1864 & T8 & (E26 + E27) & A4039, 3: ST_CON
         IF $IN[1864] AND $TIMER_FLAG[8] AND ($IN[26] OR $IN[27]) AND $OUT[4039] THEN
            PREVSTEP = $APP_INT[5]
            $APP_INT[5] = 158
         ENDIF
      ;ENDFOLD
      ;FOLD Schritt 161 = !E1864 & A4039 ;%{SE}%MKUKATPVW %CVW_SPS %VST_CON %P 2:Schritt 161 = !E1864 & A4039, 3: ST_CON
         IF NOT $IN[1864] AND $OUT[4039] THEN
            PREVSTEP = $APP_INT[5]
            $APP_INT[5] = 161
         ENDIF
      ;ENDFOLD
   ;ENDFOLD
   ;FOLD SCHRITT 161 --MS1 Reinigung (an Pneum. Schwenkeinheit MS1)-- ;%{P}%MKUKATPVW,%CSTEP,%VST_NR,%P 1:SCHRITT, 2:161, 3:MS1 Reinigung (an Pneum. Schwenkeinheit MS1)
      ;FOLD ;%{H}
         Case 161
      ;ENDFOLD
      ;FOLD -- Steuerluft EIN -- ;%{SE}%MKUKATPVW %CVW_COM %VCOMMENT %P 2:-- Steuerluft EIN --, 3: VW_COMMENT
      ;ENDFOLD
      ;FOLD A2161 = A4039 ;%{SE}%MKUKATPVW %CVW_SPS %VBOASG %P 2:A2161 = A4039, 3: BOASG
         $OUT[2161] = $OUT[4039]
      ;ENDFOLD
      ;FOLD Schritt 158 = E1864 & T9 & (E26 + E27) & A4039 ;%{SE}%MKUKATPVW %CVW_SPS %VST_CON %P 2:Schritt 158 = E1864 & T9 & (E26 + E27) & A4039, 3: ST_CON
         IF $IN[1864] AND $TIMER_FLAG[9] AND ($IN[26] OR $IN[27]) AND $OUT[4039] THEN
            PREVSTEP = $APP_INT[5]
            $APP_INT[5] = 158
         ENDIF
      ;ENDFOLD
      ;FOLD Schritt 162 = T9 & A4039 ;%{SE}%MKUKATPVW %CVW_SPS %VST_CON %P 2:Schritt 162 = T9 & A4039, 3: ST_CON
         IF $TIMER_FLAG[9] AND $OUT[4039] THEN
            PREVSTEP = $APP_INT[5]
            $APP_INT[5] = 162
         ENDIF
      ;ENDFOLD
   ;ENDFOLD
   ;FOLD SCHRITT 162 --MS1 Reinigung (an Pneum. Schwenkeinheit MS1)-- ;%{P}%MKUKATPVW,%CSTEP,%VST_NR,%P 1:SCHRITT, 2:162, 3:MS1 Reinigung (an Pneum. Schwenkeinheit MS1)
      ;FOLD ;%{H}
         Case 162
      ;ENDFOLD
      ;FOLD -- Steuerluft EIN -- ;%{SE}%MKUKATPVW %CVW_COM %VCOMMENT %P 2:-- Steuerluft EIN --, 3: VW_COMMENT
      ;ENDFOLD
      ;FOLD A2161 = A4039 ;%{SE}%MKUKATPVW %CVW_SPS %VBOASG %P 2:A2161 = A4039, 3: BOASG
         $OUT[2161] = $OUT[4039]
      ;ENDFOLD
      ;FOLD -- RSK Sammelstoerung -- ;%{SE}%MKUKATPVW %CVW_COM %VCOMMENT %P 2:-- RSK Sammelstoerung --, 3: VW_COMMENT
      ;ENDFOLD
      ;FOLD F329 = T8 ;%{SE}%MKUKATPVW %CVW_SPS %VBOASG %P 2:F329 = T8, 3: BOASG
         $FLAG[329] = $TIMER_FLAG[8]
      ;ENDFOLD
      ;FOLD -- MS1 Reinigung beenden -- ;%{SE}%MKUKATPVW %CVW_COM %VCOMMENT %P 2:-- MS1 Reinigung beenden --, 3: VW_COMMENT
      ;ENDFOLD
      ;FOLD A1864 = AUS ;%{SE}%MKUKATPVW %CVW_SPS %VBOASG %P 2:A1864 = AUS, 3: BOASG
         $OUT[1864] = FALSE
      ;ENDFOLD
      ;FOLD -- MS1 Ausblasen AUS -- ;%{SE}%MKUKATPVW %CVW_COM %VCOMMENT %P 2:-- MS1 Ausblasen AUS --, 3: VW_COMMENT
      ;ENDFOLD
      ;FOLD A1870 = AUS ;%{SE}%MKUKATPVW %CVW_SPS %VBOASG %P 2:A1870 = AUS, 3: BOASG
         $OUT[1870] = FALSE
      ;ENDFOLD
      ;FOLD -- MS1 Einspruehen EIN -- ;%{SE}%MKUKATPVW %CVW_COM %VCOMMENT %P 2:-- MS1 Einspruehen EIN --, 3: VW_COMMENT
      ;ENDFOLD
      ;FOLD A520 = !F574 & F575 ;%{SE}%MKUKATPVW %CVW_SPS %VBOASG %P 2:A520 = !F574 & F575, 3: BOASG
         $OUT[520] = NOT $FLAG[574] AND $FLAG[575]
      ;ENDFOLD
      ;FOLD A1871 = F574 & F575 ;%{SE}%MKUKATPVW %CVW_SPS %VBOASG %P 2:A1871 = F574 & F575, 3: BOASG
         $OUT[1871] = $FLAG[574] AND $FLAG[575]
      ;ENDFOLD
      ;FOLD -- Einschaltdauer Einspruehen -- ;%{SE}%MKUKATPVW %CVW_COM %VCOMMENT %P 2:-- Einschaltdauer Einspruehen --, 3: VW_COMMENT
      ;ENDFOLD
      ;FOLD t7 ( EIN ) = i23[1/10Sek] ;%{SE}%MKUKATPVW %CVW_SPS %VTASG %P 2:t7 ( EIN ) = i23[1/10Sek], 3: TASG
         VW(#SET_TIME,TRUE,7,0,$COUNT_I[23])
      ;ENDFOLD
      ;FOLD Schritt 163 = E1864 & A4039 ;%{SE}%MKUKATPVW %CVW_SPS %VST_CON %P 2:Schritt 163 = E1864 & A4039, 3: ST_CON
         IF $IN[1864] AND $OUT[4039] THEN
            PREVSTEP = $APP_INT[5]
            $APP_INT[5] = 163
         ENDIF
      ;ENDFOLD
   ;ENDFOLD
   ;FOLD SCHRITT 163 --MS1 Reinigung (an Pneum. Schwenkeinheit MS1)-- ;%{P}%MKUKATPVW,%CSTEP,%VST_NR,%P 1:SCHRITT, 2:163, 3:MS1 Reinigung (an Pneum. Schwenkeinheit MS1)
      ;FOLD ;%{H}
         Case 163
      ;ENDFOLD
      ;FOLD F323 = AUS ;%{SE}%MKUKATPVW %CVW_SPS %VBOASG %P 2:F323 = AUS, 3: BOASG
         $FLAG[323] = FALSE
      ;ENDFOLD
      ;FOLD A2163 = AUS ;%{SE}%MKUKATPVW %CVW_SPS %VBOASG %P 2:A2163 = AUS, 3: BOASG
         $OUT[2163] = FALSE
      ;ENDFOLD
      ;FOLD A2164 = AUS ;%{SE}%MKUKATPVW %CVW_SPS %VBOASG %P 2:A2164 = AUS, 3: BOASG
         $OUT[2164] = FALSE
      ;ENDFOLD
      ;FOLD A2165 = AUS ;%{SE}%MKUKATPVW %CVW_SPS %VBOASG %P 2:A2165 = AUS, 3: BOASG
         $OUT[2165] = FALSE
      ;ENDFOLD
      ;FOLD A2166 = AUS ;%{SE}%MKUKATPVW %CVW_SPS %VBOASG %P 2:A2166 = AUS, 3: BOASG
         $OUT[2166] = FALSE
      ;ENDFOLD
      ;FOLD A2168 = AUS ;%{SE}%MKUKATPVW %CVW_SPS %VBOASG %P 2:A2168 = AUS, 3: BOASG
         $OUT[2168] = FALSE
      ;ENDFOLD
      ;FOLD -- Ueberwachungszeit Schwenkeinheit 1 schwenken -- ;%{SE}%MKUKATPVW %CVW_COM %VCOMMENT %P 2:-- Ueberwachungszeit Schwenkeinheit 1 schwenken --, 3: VW_COMMENT
      ;ENDFOLD
      ;FOLD t8 ( EIN ) = -100[1/10Sek] ;%{SE}%MKUKATPVW %CVW_SPS %VTASG %P 2:t8 ( EIN ) = -100[1/10Sek], 3: TASG
         VW(#SET_TIME,TRUE,8,0,-100)
      ;ENDFOLD
      ;FOLD Schritt 164 = T7 & A4039 ;%{SE}%MKUKATPVW %CVW_SPS %VST_CON %P 2:Schritt 164 = T7 & A4039, 3: ST_CON
         IF $TIMER_FLAG[7] AND $OUT[4039] THEN
            PREVSTEP = $APP_INT[5]
            $APP_INT[5] = 164
         ENDIF
      ;ENDFOLD
   ;ENDFOLD
   ;FOLD SCHRITT 164 --MS1 Reinigung (an Pneum. Schwenkeinheit MS1)-- ;%{P}%MKUKATPVW,%CSTEP,%VST_NR,%P 1:SCHRITT, 2:164, 3:MS1 Reinigung (an Pneum. Schwenkeinheit MS1)
      ;FOLD ;%{H}
         Case 164
      ;ENDFOLD
      ;FOLD -- Steuerluft EIN -- ;%{SE}%MKUKATPVW %CVW_COM %VCOMMENT %P 2:-- Steuerluft EIN --, 3: VW_COMMENT
      ;ENDFOLD
      ;FOLD A2161 = A4039 ;%{SE}%MKUKATPVW %CVW_SPS %VBOASG %P 2:A2161 = A4039, 3: BOASG
         $OUT[2161] = $OUT[4039]
      ;ENDFOLD
      ;FOLD -- MS1 Einspruehen AUS -- ;%{SE}%MKUKATPVW %CVW_COM %VCOMMENT %P 2:-- MS1 Einspruehen AUS --, 3: VW_COMMENT
      ;ENDFOLD
      ;FOLD A520 = AUS ;%{SE}%MKUKATPVW %CVW_SPS %VBOASG %P 2:A520 = AUS, 3: BOASG
         $OUT[520] = FALSE
      ;ENDFOLD
      ;FOLD A1871 = AUS ;%{SE}%MKUKATPVW %CVW_SPS %VBOASG %P 2:A1871 = AUS, 3: BOASG
         $OUT[1871] = FALSE
      ;ENDFOLD
      ;FOLD -- Versetzeinheit in Ruhest. schw. -- ;%{SE}%MKUKATPVW %CVW_COM %VCOMMENT %P 2:-- Versetzeinheit in Ruhest. schw. --, 3: VW_COMMENT
      ;ENDFOLD
      ;FOLD A2167 = EIN ;%{SE}%MKUKATPVW %CVW_SPS %VBOASG %P 2:A2167 = EIN, 3: BOASG
         $OUT[2167] = TRUE
      ;ENDFOLD
      ;FOLD A2168 = AUS ;%{SE}%MKUKATPVW %CVW_SPS %VBOASG %P 2:A2168 = AUS, 3: BOASG
         $OUT[2168] = FALSE
      ;ENDFOLD
      ;FOLD -- RSK Fehlerausgabe Versetzeinheit in Ruhest. schw. -- ;%{SE}%MKUKATPVW %CVW_COM %VCOMMENT %P 2:-- RSK Fehlerausgabe Versetzeinheit in Ruhest. schw. --, 3: VW_COMMENT
      ;ENDFOLD
      ;FOLD F328 = F576 & T8 ;%{SE}%MKUKATPVW %CVW_SPS %VBOASG %P 2:F328 = F576 & T8, 3: BOASG
         $FLAG[328] = $FLAG[576] AND $TIMER_FLAG[8]
      ;ENDFOLD
      ;FOLD -- RSK Fehlerausgabe Schwenkeinheit 1 Arbeit. -- ;%{SE}%MKUKATPVW %CVW_COM %VCOMMENT %P 2:-- RSK Fehlerausgabe Schwenkeinheit 1 Arbeit. --, 3: VW_COMMENT
      ;ENDFOLD
      ;FOLD F324 = !E2164 & T8 ;%{SE}%MKUKATPVW %CVW_SPS %VBOASG %P 2:F324 = !E2164 & T8, 3: BOASG
         $FLAG[324] = NOT $IN[2164] AND $TIMER_FLAG[8]
      ;ENDFOLD
      ;FOLD -- RSK Sammelstoerung -- ;%{SE}%MKUKATPVW %CVW_COM %VCOMMENT %P 2:-- RSK Sammelstoerung --, 3: VW_COMMENT
      ;ENDFOLD
      ;FOLD F329 = F324 + F328 ;%{SE}%MKUKATPVW %CVW_SPS %VBOASG %P 2:F329 = F324 + F328, 3: BOASG
         $FLAG[329] = $FLAG[324] OR $FLAG[328]
      ;ENDFOLD
      ;FOLD Schritt 163 = (E26 + E27) & (F324 + F328) & A4039 ;%{SE}%MKUKATPVW %CVW_SPS %VST_CON %P 2:Schritt 163 = (E26 + E27) & (F324 + F328) & A4039, 3: ST_CON
         IF ($IN[26] OR $IN[27]) AND ($FLAG[324] OR $FLAG[328]) AND $OUT[4039] THEN
            PREVSTEP = $APP_INT[5]
            $APP_INT[5] = 163
         ENDIF
      ;ENDFOLD
      ;FOLD Schritt 165 = (!F324 + T8) & (F523 & !F524 & E2161 + !F523 & F524 & !E2162) & E2167 & F576 & A4039 ;%{SE}%MKUKATPVW %CVW_SPS %VST_CON %P 2:Schritt 165 = (!F324 + T8) & (F523 & !F524 & E2161 + !F523 & F524 & !E2162) & E2167 & F576 & A4039, 3: ST_CON
         IF (NOT $FLAG[324] OR $TIMER_FLAG[8]) AND ($FLAG[523] AND NOT $FLAG[524] AND $IN[2161] OR NOT $FLAG[523] AND $FLAG[524] AND NOT $IN[2162]) AND $IN[2167] AND $FLAG[576] AND $OUT[4039] THEN
            PREVSTEP = $APP_INT[5]
            $APP_INT[5] = 165
         ENDIF
      ;ENDFOLD
      ;FOLD Schritt 165 = (!F324 + T8) & (F523 & !F524 & E2161 + !F523 & F524 & !E2162) & !E2167 & !F576 & A4039 ;%{SE}%MKUKATPVW %CVW_SPS %VST_CON %P 2:Schritt 165 = (!F324 + T8) & (F523 & !F524 & E2161 + !F523 & F524 & !E2162) & !E2167 & !F576 & A4039, 3: ST_CON
         IF (NOT $FLAG[324] OR $TIMER_FLAG[8]) AND ($FLAG[523] AND NOT $FLAG[524] AND $IN[2161] OR NOT $FLAG[523] AND $FLAG[524] AND NOT $IN[2162]) AND NOT $IN[2167] AND NOT $FLAG[576] AND $OUT[4039] THEN
            PREVSTEP = $APP_INT[5]
            $APP_INT[5] = 165
         ENDIF
      ;ENDFOLD
   ;ENDFOLD
   ;FOLD SCHRITT 165 --MS1 Reinigung (an Pneum. Schwenkeinheit MS1)-- ;%{P}%MKUKATPVW,%CSTEP,%VST_NR,%P 1:SCHRITT, 2:165, 3:MS1 Reinigung (an Pneum. Schwenkeinheit MS1)
      ;FOLD ;%{H}
         Case 165
      ;ENDFOLD
      ;FOLD -- Steuerluft EIN -- ;%{SE}%MKUKATPVW %CVW_COM %VCOMMENT %P 2:-- Steuerluft EIN --, 3: VW_COMMENT
      ;ENDFOLD
      ;FOLD A2161 = A4039 ;%{SE}%MKUKATPVW %CVW_SPS %VBOASG %P 2:A2161 = A4039, 3: BOASG
         $OUT[2161] = $OUT[4039]
      ;ENDFOLD
      ;FOLD A2167 = AUS ;%{SE}%MKUKATPVW %CVW_SPS %VBOASG %P 2:A2167 = AUS, 3: BOASG
         $OUT[2167] = FALSE
      ;ENDFOLD
      ;FOLD -- Schwenkeinheit 1 in Ruhestellung schwenken -- ;%{SE}%MKUKATPVW %CVW_COM %VCOMMENT %P 2:-- Schwenkeinheit 1 in Ruhestellung schwenken --, 3: VW_COMMENT
      ;ENDFOLD
      ;FOLD A2163 = !E2163 ;%{SE}%MKUKATPVW %CVW_SPS %VBOASG %P 2:A2163 = !E2163, 3: BOASG
         $OUT[2163] = NOT $IN[2163]
      ;ENDFOLD
      ;FOLD A2164 = AUS ;%{SE}%MKUKATPVW %CVW_SPS %VBOASG %P 2:A2164 = AUS, 3: BOASG
         $OUT[2164] = FALSE
      ;ENDFOLD
      ;FOLD -- FRG Bewegung EIN -- ;%{SE}%MKUKATPVW %CVW_COM %VCOMMENT %P 2:-- FRG Bewegung EIN --, 3: VW_COMMENT
      ;ENDFOLD
      ;FOLD A2165 = AUS ;%{SE}%MKUKATPVW %CVW_SPS %VBOASG %P 2:A2165 = AUS, 3: BOASG
         $OUT[2165] = FALSE
      ;ENDFOLD
      ;FOLD A2166 = !E2163 ;%{SE}%MKUKATPVW %CVW_SPS %VBOASG %P 2:A2166 = !E2163, 3: BOASG
         $OUT[2166] = NOT $IN[2163]
      ;ENDFOLD
      ;FOLD Schritt 166 = E1864 & !E2164 & E2163 & A4039 + T8 ;%{SE}%MKUKATPVW %CVW_SPS %VST_CON %P 2:Schritt 166 = E1864 & !E2164 & E2163 & A4039 + T8, 3: ST_CON
         IF $IN[1864] AND NOT $IN[2164] AND $IN[2163] AND $OUT[4039] OR $TIMER_FLAG[8] THEN
            PREVSTEP = $APP_INT[5]
            $APP_INT[5] = 166
         ENDIF
      ;ENDFOLD
   ;ENDFOLD
   ;FOLD SCHRITT 166 --MS1 Reinigung (an Pneum. Schwenkeinheit MS1)-- ;%{P}%MKUKATPVW,%CSTEP,%VST_NR,%P 1:SCHRITT, 2:166, 3:MS1 Reinigung (an Pneum. Schwenkeinheit MS1)
      ;FOLD ;%{H}
         Case 166
      ;ENDFOLD
      ;FOLD -- Steuerluft EIN -- ;%{SE}%MKUKATPVW %CVW_COM %VCOMMENT %P 2:-- Steuerluft EIN --, 3: VW_COMMENT
      ;ENDFOLD
      ;FOLD A2161 = A4039 ;%{SE}%MKUKATPVW %CVW_SPS %VBOASG %P 2:A2161 = A4039, 3: BOASG
         $OUT[2161] = $OUT[4039]
      ;ENDFOLD
      ;FOLD -- RSK Fehlerausgabe Schwenkeinheit 1 Ruhestellung -- ;%{SE}%MKUKATPVW %CVW_COM %VCOMMENT %P 2:-- RSK Fehlerausgabe Schwenkeinheit 1 Ruhestellung --, 3: VW_COMMENT
      ;ENDFOLD
      ;FOLD F323 = !E2163 & T8 + F323 ;%{SE}%MKUKATPVW %CVW_SPS %VBOASG %P 2:F323 = !E2163 & T8 + F323, 3: BOASG
         $FLAG[323] = NOT $IN[2163] AND $TIMER_FLAG[8] OR $FLAG[323]
      ;ENDFOLD
      ;FOLD -- RSK Sammelstoerung -- ;%{SE}%MKUKATPVW %CVW_COM %VCOMMENT %P 2:-- RSK Sammelstoerung --, 3: VW_COMMENT
      ;ENDFOLD
      ;FOLD F329 = F323 ;%{SE}%MKUKATPVW %CVW_SPS %VBOASG %P 2:F329 = F323, 3: BOASG
         $FLAG[329] = $FLAG[323]
      ;ENDFOLD
      ;FOLD A2163 = AUS ;%{SE}%MKUKATPVW %CVW_SPS %VBOASG %P 2:A2163 = AUS, 3: BOASG
         $OUT[2163] = FALSE
      ;ENDFOLD
      ;FOLD -- FRG Bewegung AUS -- ;%{SE}%MKUKATPVW %CVW_COM %VCOMMENT %P 2:-- FRG Bewegung AUS --, 3: VW_COMMENT
      ;ENDFOLD
      ;FOLD A2166 = AUS ;%{SE}%MKUKATPVW %CVW_SPS %VBOASG %P 2:A2166 = AUS, 3: BOASG
         $OUT[2166] = FALSE
      ;ENDFOLD
      ;FOLD Schritt 163 = F323 & (E26 + E27) & A4039 ;%{SE}%MKUKATPVW %CVW_SPS %VST_CON %P 2:Schritt 163 = F323 & (E26 + E27) & A4039, 3: ST_CON
         IF $FLAG[323] AND ($IN[26] OR $IN[27]) AND $OUT[4039] THEN
            PREVSTEP = $APP_INT[5]
            $APP_INT[5] = 163
         ENDIF
      ;ENDFOLD
      ;FOLD Schritt 167 = !F323 & E2166 & A4039 ;%{SE}%MKUKATPVW %CVW_SPS %VST_CON %P 2:Schritt 167 = !F323 & E2166 & A4039, 3: ST_CON
         IF NOT $FLAG[323] AND $IN[2166] AND $OUT[4039] THEN
            PREVSTEP = $APP_INT[5]
            $APP_INT[5] = 167
         ENDIF
      ;ENDFOLD
   ;ENDFOLD
   ;FOLD SCHRITT 167 --MS1 Reinigung (an Pneum. Schwenkeinheit MS1)-- ;%{P}%MKUKATPVW,%CSTEP,%VST_NR,%P 1:SCHRITT, 2:167, 3:MS1 Reinigung (an Pneum. Schwenkeinheit MS1)
      ;FOLD ;%{H}
         Case 167
      ;ENDFOLD
      ;FOLD -- Steuerluft EIN -- ;%{SE}%MKUKATPVW %CVW_COM %VCOMMENT %P 2:-- Steuerluft EIN --, 3: VW_COMMENT
      ;ENDFOLD
      ;FOLD A2161 = A4039 ;%{SE}%MKUKATPVW %CVW_SPS %VBOASG %P 2:A2161 = A4039, 3: BOASG
         $OUT[2161] = $OUT[4039]
      ;ENDFOLD
      ;FOLD -- RSK Sammelstoerung -- ;%{SE}%MKUKATPVW %CVW_COM %VCOMMENT %P 2:-- RSK Sammelstoerung --, 3: VW_COMMENT
      ;ENDFOLD
      ;FOLD F329 = T8 ;%{SE}%MKUKATPVW %CVW_SPS %VBOASG %P 2:F329 = T8, 3: BOASG
         $FLAG[329] = $TIMER_FLAG[8]
      ;ENDFOLD
      ;FOLD F323 = AUS ;%{SE}%MKUKATPVW %CVW_SPS %VBOASG %P 2:F323 = AUS, 3: BOASG
         $FLAG[323] = FALSE
      ;ENDFOLD
      ;FOLD -- FRG in Endlage halten ein -- ;%{SE}%MKUKATPVW %CVW_COM %VCOMMENT %P 2:-- FRG in Endlage halten ein --, 3: VW_COMMENT
      ;ENDFOLD
      ;FOLD A2165 = EIN ;%{SE}%MKUKATPVW %CVW_SPS %VBOASG %P 2:A2165 = EIN, 3: BOASG
         $OUT[2165] = TRUE
      ;ENDFOLD
      ;FOLD Schritt 168 = E2165 & A4039 ;%{SE}%MKUKATPVW %CVW_SPS %VST_CON %P 2:Schritt 168 = E2165 & A4039, 3: ST_CON
         IF $IN[2165] AND $OUT[4039] THEN
            PREVSTEP = $APP_INT[5]
            $APP_INT[5] = 168
         ENDIF
      ;ENDFOLD
   ;ENDFOLD
   ;FOLD SCHRITT 168 --MS1 Reinigung (an Pneum. Schwenkeinheit MS1)-- ;%{P}%MKUKATPVW,%CSTEP,%VST_NR,%P 1:SCHRITT, 2:168, 3:MS1 Reinigung (an Pneum. Schwenkeinheit MS1)
      ;FOLD ;%{H}
         Case 168
      ;ENDFOLD
      ;FOLD -- Steuerluft EIN -- ;%{SE}%MKUKATPVW %CVW_COM %VCOMMENT %P 2:-- Steuerluft EIN --, 3: VW_COMMENT
      ;ENDFOLD
      ;FOLD A2161 = A4039 ;%{SE}%MKUKATPVW %CVW_SPS %VBOASG %P 2:A2161 = A4039, 3: BOASG
         $OUT[2161] = $OUT[4039]
      ;ENDFOLD
      ;FOLD -- FRG in Endlage halten AUS -- ;%{SE}%MKUKATPVW %CVW_COM %VCOMMENT %P 2:-- FRG in Endlage halten AUS --, 3: VW_COMMENT
      ;ENDFOLD
      ;FOLD A2165 = AUS ;%{SE}%MKUKATPVW %CVW_SPS %VBOASG %P 2:A2165 = AUS, 3: BOASG
         $OUT[2165] = FALSE
      ;ENDFOLD
      ;FOLD -- MS1 Zaehler ruecksetzen -- ;%{SE}%MKUKATPVW %CVW_COM %VCOMMENT %P 2:-- MS1 Zaehler ruecksetzen --, 3: VW_COMMENT
      ;ENDFOLD
      ;FOLD -- MS1 FRG Reinigung -- ;%{SE}%MKUKATPVW %CVW_COM %VCOMMENT %P 2:-- MS1 FRG Reinigung --, 3: VW_COMMENT
      ;ENDFOLD
      ;FOLD F603 = AUS ;%{SE}%MKUKATPVW %CVW_SPS %VBOASG %P 2:F603 = AUS, 3: BOASG
         $FLAG[603] = FALSE
      ;ENDFOLD
      ;FOLD -- MS1 Reinigung FK -- ;%{SE}%MKUKATPVW %CVW_COM %VCOMMENT %P 2:-- MS1 Reinigung FK --, 3: VW_COMMENT
      ;ENDFOLD
      ;FOLD F605 = EIN ;%{SE}%MKUKATPVW %CVW_SPS %VBOASG %P 2:F605 = EIN, 3: BOASG
         $FLAG[605] = TRUE
      ;ENDFOLD
      ;FOLD t8 ( EIN ) = STOP ;%{SE}%MKUKATPVW %CVW_SPS %VTSTOP %P 2:t8 ( EIN ) = STOP, 3: TSTOP
         VW(#SET_TIME,TRUE,8,1,0)
      ;ENDFOLD
      ;FOLD Schritt 1 = A4039 ;%{SE}%MKUKATPVW %CVW_SPS %VST_CON %P 2:Schritt 1 = A4039, 3: ST_CON
         IF $OUT[4039] THEN
            PREVSTEP = $APP_INT[5]
            $APP_INT[5] = 1
         ENDIF
      ;ENDFOLD
   ;ENDFOLD
   ;FOLD SCHRITT 169 --MS2 Reinigung (an Pneum. Schwenkeinheit MS2)-- ;%{P}%MKUKATPVW,%CSTEP,%VST_NR,%P 1:SCHRITT, 2:169, 3:MS2 Reinigung (an Pneum. Schwenkeinheit MS2)
      ;FOLD ;%{H}
         Case 169
      ;ENDFOLD
      ;FOLD -- RSK gestartet -- ;%{SE}%MKUKATPVW %CVW_COM %VCOMMENT %P 2:-- RSK gestartet --, 3: VW_COMMENT
      ;ENDFOLD
      ;FOLD F321 = AUS ;%{SE}%MKUKATPVW %CVW_SPS %VBOASG %P 2:F321 = AUS, 3: BOASG
         $FLAG[321] = FALSE
      ;ENDFOLD
      ;FOLD F323 = AUS ;%{SE}%MKUKATPVW %CVW_SPS %VBOASG %P 2:F323 = AUS, 3: BOASG
         $FLAG[323] = FALSE
      ;ENDFOLD
      ;FOLD F324 = AUS ;%{SE}%MKUKATPVW %CVW_SPS %VBOASG %P 2:F324 = AUS, 3: BOASG
         $FLAG[324] = FALSE
      ;ENDFOLD
      ;FOLD F329 = AUS ;%{SE}%MKUKATPVW %CVW_SPS %VBOASG %P 2:F329 = AUS, 3: BOASG
         $FLAG[329] = FALSE
      ;ENDFOLD
      ;FOLD -- MS2 Reinigung gestartet -- ;%{SE}%MKUKATPVW %CVW_COM %VCOMMENT %P 2:-- MS2 Reinigung gestartet --, 3: VW_COMMENT
      ;ENDFOLD
      ;FOLD F608 = EIN ;%{SE}%MKUKATPVW %CVW_SPS %VBOASG %P 2:F608 = EIN, 3: BOASG
         $FLAG[608] = TRUE
      ;ENDFOLD
      ;FOLD -- Steuerluft EIN -- ;%{SE}%MKUKATPVW %CVW_COM %VCOMMENT %P 2:-- Steuerluft EIN --, 3: VW_COMMENT
      ;ENDFOLD
      ;FOLD A2169 = A4039 ;%{SE}%MKUKATPVW %CVW_SPS %VBOASG %P 2:A2169 = A4039, 3: BOASG
         $OUT[2169] = $OUT[4039]
      ;ENDFOLD
      ;FOLD A2171 = AUS ;%{SE}%MKUKATPVW %CVW_SPS %VBOASG %P 2:A2171 = AUS, 3: BOASG
         $OUT[2171] = FALSE
      ;ENDFOLD
      ;FOLD A2172 = AUS ;%{SE}%MKUKATPVW %CVW_SPS %VBOASG %P 2:A2172 = AUS, 3: BOASG
         $OUT[2172] = FALSE
      ;ENDFOLD
      ;FOLD A2173 = AUS ;%{SE}%MKUKATPVW %CVW_SPS %VBOASG %P 2:A2173 = AUS, 3: BOASG
         $OUT[2173] = FALSE
      ;ENDFOLD
      ;FOLD A2174 = AUS ;%{SE}%MKUKATPVW %CVW_SPS %VBOASG %P 2:A2174 = AUS, 3: BOASG
         $OUT[2174] = FALSE
      ;ENDFOLD
      ;FOLD A2175 = AUS ;%{SE}%MKUKATPVW %CVW_SPS %VBOASG %P 2:A2175 = AUS, 3: BOASG
         $OUT[2175] = FALSE
      ;ENDFOLD
      ;FOLD A2176 = AUS ;%{SE}%MKUKATPVW %CVW_SPS %VBOASG %P 2:A2176 = AUS, 3: BOASG
         $OUT[2176] = FALSE
      ;ENDFOLD
      ;FOLD -- Ueberwachungszeit Schwenkeinheit 2 -- ;%{SE}%MKUKATPVW %CVW_COM %VCOMMENT %P 2:-- Ueberwachungszeit Schwenkeinheit 2 --, 3: VW_COMMENT
      ;ENDFOLD
      ;FOLD t8 ( EIN ) = -100[1/10Sek] ;%{SE}%MKUKATPVW %CVW_SPS %VTASG %P 2:t8 ( EIN ) = -100[1/10Sek], 3: TASG
         VW(#SET_TIME,TRUE,8,0,-100)
      ;ENDFOLD
      ;FOLD Schritt 170 = A4039 ;%{SE}%MKUKATPVW %CVW_SPS %VST_CON %P 2:Schritt 170 = A4039, 3: ST_CON
         IF $OUT[4039] THEN
            PREVSTEP = $APP_INT[5]
            $APP_INT[5] = 170
         ENDIF
      ;ENDFOLD
   ;ENDFOLD
   ;FOLD SCHRITT 170 --MS2 Reinigung (an Pneum. Schwenkeinheit MS2)-- ;%{P}%MKUKATPVW,%CSTEP,%VST_NR,%P 1:SCHRITT, 2:170, 3:MS2 Reinigung (an Pneum. Schwenkeinheit MS2)
      ;FOLD ;%{H}
         Case 170
      ;ENDFOLD
      ;FOLD -- Steuerluft EIN -- ;%{SE}%MKUKATPVW %CVW_COM %VCOMMENT %P 2:-- Steuerluft EIN --, 3: VW_COMMENT
      ;ENDFOLD
      ;FOLD A2169 = A4039 ;%{SE}%MKUKATPVW %CVW_SPS %VBOASG %P 2:A2169 = A4039, 3: BOASG
         $OUT[2169] = $OUT[4039]
      ;ENDFOLD
      ;FOLD -- RSK Fehlerausgabe Schwenkeinheit 2 Ruhest. -- ;%{SE}%MKUKATPVW %CVW_COM %VCOMMENT %P 2:-- RSK Fehlerausgabe Schwenkeinheit 2 Ruhest. --, 3: VW_COMMENT
      ;ENDFOLD
      ;FOLD F323 = !E2171 & T8 ;%{SE}%MKUKATPVW %CVW_SPS %VBOASG %P 2:F323 = !E2171 & T8, 3: BOASG
         $FLAG[323] = NOT $IN[2171] AND $TIMER_FLAG[8]
      ;ENDFOLD
      ;FOLD -- RSK Sammelstoerung -- ;%{SE}%MKUKATPVW %CVW_COM %VCOMMENT %P 2:-- RSK Sammelstoerung --, 3: VW_COMMENT
      ;ENDFOLD
      ;FOLD F329 = F323 + T8 ;%{SE}%MKUKATPVW %CVW_SPS %VBOASG %P 2:F329 = F323 + T8, 3: BOASG
         $FLAG[329] = $FLAG[323] OR $TIMER_FLAG[8]
      ;ENDFOLD
      ;FOLD Schritt 169 = (E26 + E27) & F323 & A4039 ;%{SE}%MKUKATPVW %CVW_SPS %VST_CON %P 2:Schritt 169 = (E26 + E27) & F323 & A4039, 3: ST_CON
         IF ($IN[26] OR $IN[27]) AND $FLAG[323] AND $OUT[4039] THEN
            PREVSTEP = $APP_INT[5]
            $APP_INT[5] = 169
         ENDIF
      ;ENDFOLD
      ;FOLD Schritt 171 = (!F323 + T8) & (F523 & !F524 & E2169 + !F523 & F524 & !E2170) & A4039 ;%{SE}%MKUKATPVW %CVW_SPS %VST_CON %P 2:Schritt 171 = (!F323 + T8) & (F523 & !F524 & E2169 + !F523 & F524 & !E2170) & A4039, 3: ST_CON
         IF (NOT $FLAG[323] OR $TIMER_FLAG[8]) AND ($FLAG[523] AND NOT $FLAG[524] AND $IN[2169] OR NOT $FLAG[523] AND $FLAG[524] AND NOT $IN[2170]) AND $OUT[4039] THEN
            PREVSTEP = $APP_INT[5]
            $APP_INT[5] = 171
         ENDIF
      ;ENDFOLD
   ;ENDFOLD
   ;FOLD SCHRITT 171 --MS2 Reinigung (an Pneum. Schwenkeinheit MS2)-- ;%{P}%MKUKATPVW,%CSTEP,%VST_NR,%P 1:SCHRITT, 2:171, 3:MS2 Reinigung (an Pneum. Schwenkeinheit MS2)
      ;FOLD ;%{H}
         Case 171
      ;ENDFOLD
      ;FOLD -- Steuerluft EIN -- ;%{SE}%MKUKATPVW %CVW_COM %VCOMMENT %P 2:-- Steuerluft EIN --, 3: VW_COMMENT
      ;ENDFOLD
      ;FOLD A2169 = A4039 ;%{SE}%MKUKATPVW %CVW_SPS %VBOASG %P 2:A2169 = A4039, 3: BOASG
         $OUT[2169] = $OUT[4039]
      ;ENDFOLD
      ;FOLD -- Schwenkeinheit 2 in Arbeitsstellung schwenken -- ;%{SE}%MKUKATPVW %CVW_COM %VCOMMENT %P 2:-- Schwenkeinheit 2 in Arbeitsstellung schwenken --, 3: VW_COMMENT
      ;ENDFOLD
      ;FOLD A2172 = EIN ;%{SE}%MKUKATPVW %CVW_SPS %VBOASG %P 2:A2172 = EIN, 3: BOASG
         $OUT[2172] = TRUE
      ;ENDFOLD
      ;FOLD -- FRG Bewegung EIN -- ;%{SE}%MKUKATPVW %CVW_COM %VCOMMENT %P 2:-- FRG Bewegung EIN --, 3: VW_COMMENT
      ;ENDFOLD
      ;FOLD A2173 = AUS ;%{SE}%MKUKATPVW %CVW_SPS %VBOASG %P 2:A2173 = AUS, 3: BOASG
         $OUT[2173] = FALSE
      ;ENDFOLD
      ;FOLD A2174 = EIN ;%{SE}%MKUKATPVW %CVW_SPS %VBOASG %P 2:A2174 = EIN, 3: BOASG
         $OUT[2174] = TRUE
      ;ENDFOLD
      ;FOLD -- Zeit Endlage entprellen -- ;%{SE}%MKUKATPVW %CVW_COM %VCOMMENT %P 2:-- Zeit Endlage entprellen --, 3: VW_COMMENT
      ;ENDFOLD
      ;FOLD t9 ( !E2172 ) = -10[1/10Sek] ;%{SE}%MKUKATPVW %CVW_SPS %VTASG %P 2:t9 ( !E2172 ) = -10[1/10Sek], 3: TASG
         VW(#SET_TIME,NOT $IN[2172],9,0,-10)
      ;ENDFOLD
      ;FOLD Schritt 172 = E2172 & !E2171 & A4039 & T9 + T8 ;%{SE}%MKUKATPVW %CVW_SPS %VST_CON %P 2:Schritt 172 = E2172 & !E2171 & A4039 & T9 + T8, 3: ST_CON
         IF $IN[2172] AND NOT $IN[2171] AND $OUT[4039] AND $TIMER_FLAG[9] OR $TIMER_FLAG[8] THEN
            PREVSTEP = $APP_INT[5]
            $APP_INT[5] = 172
         ENDIF
      ;ENDFOLD
   ;ENDFOLD
   ;FOLD SCHRITT 172 --MS2 Reinigung (an Pneum. Schwenkeinheit MS2)-- ;%{P}%MKUKATPVW,%CSTEP,%VST_NR,%P 1:SCHRITT, 2:172, 3:MS2 Reinigung (an Pneum. Schwenkeinheit MS2)
      ;FOLD ;%{H}
         Case 172
      ;ENDFOLD
      ;FOLD -- Steuerluft EIN -- ;%{SE}%MKUKATPVW %CVW_COM %VCOMMENT %P 2:-- Steuerluft EIN --, 3: VW_COMMENT
      ;ENDFOLD
      ;FOLD A2169 = A4039 ;%{SE}%MKUKATPVW %CVW_SPS %VBOASG %P 2:A2169 = A4039, 3: BOASG
         $OUT[2169] = $OUT[4039]
      ;ENDFOLD
      ;FOLD -- RSK Fehlerausgabe Schwenkeinheit 2 Arbeitsstellung -- ;%{SE}%MKUKATPVW %CVW_COM %VCOMMENT %P 2:-- RSK Fehlerausgabe Schwenkeinheit 2 Arbeitsstellung --, 3: VW_COMMENT
      ;ENDFOLD
      ;FOLD F324 = !E2172 & T8 + F324 ;%{SE}%MKUKATPVW %CVW_SPS %VBOASG %P 2:F324 = !E2172 & T8 + F324, 3: BOASG
         $FLAG[324] = NOT $IN[2172] AND $TIMER_FLAG[8] OR $FLAG[324]
      ;ENDFOLD
      ;FOLD -- RSK Sammelstoerung -- ;%{SE}%MKUKATPVW %CVW_COM %VCOMMENT %P 2:-- RSK Sammelstoerung --, 3: VW_COMMENT
      ;ENDFOLD
      ;FOLD F329 = F324 ;%{SE}%MKUKATPVW %CVW_SPS %VBOASG %P 2:F329 = F324, 3: BOASG
         $FLAG[329] = $FLAG[324]
      ;ENDFOLD
      ;FOLD A2172 = AUS ;%{SE}%MKUKATPVW %CVW_SPS %VBOASG %P 2:A2172 = AUS, 3: BOASG
         $OUT[2172] = FALSE
      ;ENDFOLD
      ;FOLD -- FRG Bewegung AUS -- ;%{SE}%MKUKATPVW %CVW_COM %VCOMMENT %P 2:-- FRG Bewegung AUS --, 3: VW_COMMENT
      ;ENDFOLD
      ;FOLD A2174 = AUS ;%{SE}%MKUKATPVW %CVW_SPS %VBOASG %P 2:A2174 = AUS, 3: BOASG
         $OUT[2174] = FALSE
      ;ENDFOLD
      ;FOLD -- FRG in Endlage halten ein -- ;%{SE}%MKUKATPVW %CVW_COM %VCOMMENT %P 2:-- FRG in Endlage halten ein --, 3: VW_COMMENT
      ;ENDFOLD
      ;FOLD A2173 = EIN ;%{SE}%MKUKATPVW %CVW_SPS %VBOASG %P 2:A2173 = EIN, 3: BOASG
         $OUT[2173] = TRUE
      ;ENDFOLD
      ;FOLD Schritt 169 = F324 & (E26 + E27) & A4039 ;%{SE}%MKUKATPVW %CVW_SPS %VST_CON %P 2:Schritt 169 = F324 & (E26 + E27) & A4039, 3: ST_CON
         IF $FLAG[324] AND ($IN[26] OR $IN[27]) AND $OUT[4039] THEN
            PREVSTEP = $APP_INT[5]
            $APP_INT[5] = 169
         ENDIF
      ;ENDFOLD
      ;FOLD Schritt 173 = !F324 & E2172 & A4039 ;%{SE}%MKUKATPVW %CVW_SPS %VST_CON %P 2:Schritt 173 = !F324 & E2172 & A4039, 3: ST_CON
         IF NOT $FLAG[324] AND $IN[2172] AND $OUT[4039] THEN
            PREVSTEP = $APP_INT[5]
            $APP_INT[5] = 173
         ENDIF
      ;ENDFOLD
   ;ENDFOLD
   ;FOLD SCHRITT 173 --MS2 Reinigung (an Pneum. Schwenkeinheit MS2)-- ;%{P}%MKUKATPVW,%CSTEP,%VST_NR,%P 1:SCHRITT, 2:173, 3:MS2 Reinigung (an Pneum. Schwenkeinheit MS2)
      ;FOLD ;%{H}
         Case 173
      ;ENDFOLD
      ;FOLD -- Steuerluft EIN -- ;%{SE}%MKUKATPVW %CVW_COM %VCOMMENT %P 2:-- Steuerluft EIN --, 3: VW_COMMENT
      ;ENDFOLD
      ;FOLD A2169 = A4039 ;%{SE}%MKUKATPVW %CVW_SPS %VBOASG %P 2:A2169 = A4039, 3: BOASG
         $OUT[2169] = $OUT[4039]
      ;ENDFOLD
      ;FOLD A1896 = AUS ;%{SE}%MKUKATPVW %CVW_SPS %VBOASG %P 2:A1896 = AUS, 3: BOASG
         $OUT[1896] = FALSE
      ;ENDFOLD
      ;FOLD A2175 = AUS ;%{SE}%MKUKATPVW %CVW_SPS %VBOASG %P 2:A2175 = AUS, 3: BOASG
         $OUT[2175] = FALSE
      ;ENDFOLD
      ;FOLD -- Ueberwachungszeit Versetzeinheit -- ;%{SE}%MKUKATPVW %CVW_COM %VCOMMENT %P 2:-- Ueberwachungszeit Versetzeinheit --, 3: VW_COMMENT
      ;ENDFOLD
      ;FOLD t8 ( EIN ) = -100[1/10Sek] ;%{SE}%MKUKATPVW %CVW_SPS %VTASG %P 2:t8 ( EIN ) = -100[1/10Sek], 3: TASG
         VW(#SET_TIME,TRUE,8,0,-100)
      ;ENDFOLD
      ;FOLD Schritt 174 = A4039 ;%{SE}%MKUKATPVW %CVW_SPS %VST_CON %P 2:Schritt 174 = A4039, 3: ST_CON
         IF $OUT[4039] THEN
            PREVSTEP = $APP_INT[5]
            $APP_INT[5] = 174
         ENDIF
      ;ENDFOLD
   ;ENDFOLD
   ;FOLD SCHRITT 174 --MS2 Reinigung (an Pneum. Schwenkeinheit MS2)-- ;%{P}%MKUKATPVW,%CSTEP,%VST_NR,%P 1:SCHRITT, 2:174, 3:MS2 Reinigung (an Pneum. Schwenkeinheit MS2)
      ;FOLD ;%{H}
         Case 174
      ;ENDFOLD
      ;FOLD -- Steuerluft EIN -- ;%{SE}%MKUKATPVW %CVW_COM %VCOMMENT %P 2:-- Steuerluft EIN --, 3: VW_COMMENT
      ;ENDFOLD
      ;FOLD A2169 = A4039 ;%{SE}%MKUKATPVW %CVW_SPS %VBOASG %P 2:A2169 = A4039, 3: BOASG
         $OUT[2169] = $OUT[4039]
      ;ENDFOLD
      ;FOLD -- RSK Fehlerausgabe Versetzeinheit -- ;%{SE}%MKUKATPVW %CVW_COM %VCOMMENT %P 2:-- RSK Fehlerausgabe Versetzeinheit --, 3: VW_COMMENT
      ;ENDFOLD
      ;FOLD F328 = F585 & T8 ;%{SE}%MKUKATPVW %CVW_SPS %VBOASG %P 2:F328 = F585 & T8, 3: BOASG
         $FLAG[328] = $FLAG[585] AND $TIMER_FLAG[8]
      ;ENDFOLD
      ;FOLD -- RSK Sammelstoerung -- ;%{SE}%MKUKATPVW %CVW_COM %VCOMMENT %P 2:-- RSK Sammelstoerung --, 3: VW_COMMENT
      ;ENDFOLD
      ;FOLD F329 = T8 ;%{SE}%MKUKATPVW %CVW_SPS %VBOASG %P 2:F329 = T8, 3: BOASG
         $FLAG[329] = $TIMER_FLAG[8]
      ;ENDFOLD
      ;FOLD -- Versetzeinheit in Arbeitsst. schw. -- ;%{SE}%MKUKATPVW %CVW_COM %VCOMMENT %P 2:-- Versetzeinheit in Arbeitsst. schw. --, 3: VW_COMMENT
      ;ENDFOLD
      ;FOLD A2176 = !E2176 & E2172 & F585 ;%{SE}%MKUKATPVW %CVW_SPS %VBOASG %P 2:A2176 = !E2176 & E2172 & F585, 3: BOASG
         $OUT[2176] = NOT $IN[2176] AND $IN[2172] AND $FLAG[585]
      ;ENDFOLD
      ;FOLD Schritt 173 = A2176 & T8 & (E26 + E27) & A4039 ;%{SE}%MKUKATPVW %CVW_SPS %VST_CON %P 2:Schritt 173 = A2176 & T8 & (E26 + E27) & A4039, 3: ST_CON
         IF $OUT[2176] AND $TIMER_FLAG[8] AND ($IN[26] OR $IN[27]) AND $OUT[4039] THEN
            PREVSTEP = $APP_INT[5]
            $APP_INT[5] = 173
         ENDIF
      ;ENDFOLD
      ;FOLD Schritt 175 = (E2176 & F585 + !E2168 & !F585) & A4039 ;%{SE}%MKUKATPVW %CVW_SPS %VST_CON %P 2:Schritt 175 = (E2176 & F585 + !E2168 & !F585) & A4039, 3: ST_CON
         IF ($IN[2176] AND $FLAG[585] OR NOT $IN[2168] AND NOT $FLAG[585]) AND $OUT[4039] THEN
            PREVSTEP = $APP_INT[5]
            $APP_INT[5] = 175
         ENDIF
      ;ENDFOLD
   ;ENDFOLD
   ;FOLD SCHRITT 175 --MS2 Reinigung (an Pneum.  Schwenkeinheit  MS2)-- ;%{P}%MKUKATPVW,%CSTEP,%VST_NR,%P 1:SCHRITT, 2:175, 3:MS2 Reinigung (an Pneum.  Schwenkeinheit  MS2)
      ;FOLD ;%{H}
         Case 175
      ;ENDFOLD
      ;FOLD -- Steuerluft EIN -- ;%{SE}%MKUKATPVW %CVW_COM %VCOMMENT %P 2:-- Steuerluft EIN --, 3: VW_COMMENT
      ;ENDFOLD
      ;FOLD A2169 = A4039 ;%{SE}%MKUKATPVW %CVW_SPS %VBOASG %P 2:A2169 = A4039, 3: BOASG
         $OUT[2169] = $OUT[4039]
      ;ENDFOLD
      ;FOLD -- RSK Sammelstoerung -- ;%{SE}%MKUKATPVW %CVW_COM %VCOMMENT %P 2:-- RSK Sammelstoerung --, 3: VW_COMMENT
      ;ENDFOLD
      ;FOLD F329 = T8 ;%{SE}%MKUKATPVW %CVW_SPS %VBOASG %P 2:F329 = T8, 3: BOASG
         $FLAG[329] = $TIMER_FLAG[8]
      ;ENDFOLD
      ;FOLD -- Zeit Reinigung -- ;%{SE}%MKUKATPVW %CVW_COM %VCOMMENT %P 2:-- Zeit Reinigung --, 3: VW_COMMENT
      ;ENDFOLD
      ;FOLD t9 ( EIN ) = -20[1/10Sek] ;%{SE}%MKUKATPVW %CVW_SPS %VTASG %P 2:t9 ( EIN ) = -20[1/10Sek], 3: TASG
         VW(#SET_TIME,TRUE,9,0,-20)
      ;ENDFOLD
      ;FOLD -- MS2 Ausblasen EIN -- ;%{SE}%MKUKATPVW %CVW_COM %VCOMMENT %P 2:-- MS2 Ausblasen EIN --, 3: VW_COMMENT
      ;ENDFOLD
      ;FOLD A1902 = EIN ;%{SE}%MKUKATPVW %CVW_SPS %VBOASG %P 2:A1902 = EIN, 3: BOASG
         $OUT[1902] = TRUE
      ;ENDFOLD
      ;FOLD -- MS2 Reinigung starten -- ;%{SE}%MKUKATPVW %CVW_COM %VCOMMENT %P 2:-- MS2 Reinigung starten --, 3: VW_COMMENT
      ;ENDFOLD
      ;FOLD A1896 = EIN ;%{SE}%MKUKATPVW %CVW_SPS %VBOASG %P 2:A1896 = EIN, 3: BOASG
         $OUT[1896] = TRUE
      ;ENDFOLD
      ;FOLD Schritt 173 = E1896 & T8 & (E26 + E27) & A4039 ;%{SE}%MKUKATPVW %CVW_SPS %VST_CON %P 2:Schritt 173 = E1896 & T8 & (E26 + E27) & A4039, 3: ST_CON
         IF $IN[1896] AND $TIMER_FLAG[8] AND ($IN[26] OR $IN[27]) AND $OUT[4039] THEN
            PREVSTEP = $APP_INT[5]
            $APP_INT[5] = 173
         ENDIF
      ;ENDFOLD
      ;FOLD Schritt 176 = !E1896 & A4039 ;%{SE}%MKUKATPVW %CVW_SPS %VST_CON %P 2:Schritt 176 = !E1896 & A4039, 3: ST_CON
         IF NOT $IN[1896] AND $OUT[4039] THEN
            PREVSTEP = $APP_INT[5]
            $APP_INT[5] = 176
         ENDIF
      ;ENDFOLD
   ;ENDFOLD
   ;FOLD SCHRITT 176 --MS2 Reinigung (an Pneum.  Schwenkeinheit  MS2)-- ;%{P}%MKUKATPVW,%CSTEP,%VST_NR,%P 1:SCHRITT, 2:176, 3:MS2 Reinigung (an Pneum.  Schwenkeinheit  MS2)
      ;FOLD ;%{H}
         Case 176
      ;ENDFOLD
      ;FOLD -- Steuerluft EIN -- ;%{SE}%MKUKATPVW %CVW_COM %VCOMMENT %P 2:-- Steuerluft EIN --, 3: VW_COMMENT
      ;ENDFOLD
      ;FOLD A2169 = A4039 ;%{SE}%MKUKATPVW %CVW_SPS %VBOASG %P 2:A2169 = A4039, 3: BOASG
         $OUT[2169] = $OUT[4039]
      ;ENDFOLD
      ;FOLD Schritt 173 = !E1896 & T9 & (E26 + E27) & A4039 ;%{SE}%MKUKATPVW %CVW_SPS %VST_CON %P 2:Schritt 173 = !E1896 & T9 & (E26 + E27) & A4039, 3: ST_CON
         IF NOT $IN[1896] AND $TIMER_FLAG[9] AND ($IN[26] OR $IN[27]) AND $OUT[4039] THEN
            PREVSTEP = $APP_INT[5]
            $APP_INT[5] = 173
         ENDIF
      ;ENDFOLD
      ;FOLD Schritt 177 = T9 & A4039 ;%{SE}%MKUKATPVW %CVW_SPS %VST_CON %P 2:Schritt 177 = T9 & A4039, 3: ST_CON
         IF $TIMER_FLAG[9] AND $OUT[4039] THEN
            PREVSTEP = $APP_INT[5]
            $APP_INT[5] = 177
         ENDIF
      ;ENDFOLD
   ;ENDFOLD
   ;FOLD SCHRITT 177 --MS2 Reinigung (an Pneum. Schwenkeinheit MS2)-- ;%{P}%MKUKATPVW,%CSTEP,%VST_NR,%P 1:SCHRITT, 2:177, 3:MS2 Reinigung (an Pneum. Schwenkeinheit MS2)
      ;FOLD ;%{H}
         Case 177
      ;ENDFOLD
      ;FOLD -- Steuerluft EIN -- ;%{SE}%MKUKATPVW %CVW_COM %VCOMMENT %P 2:-- Steuerluft EIN --, 3: VW_COMMENT
      ;ENDFOLD
      ;FOLD A2169 = A4039 ;%{SE}%MKUKATPVW %CVW_SPS %VBOASG %P 2:A2169 = A4039, 3: BOASG
         $OUT[2169] = $OUT[4039]
      ;ENDFOLD
      ;FOLD -- RSK Sammelstoerung -- ;%{SE}%MKUKATPVW %CVW_COM %VCOMMENT %P 2:-- RSK Sammelstoerung --, 3: VW_COMMENT
      ;ENDFOLD
      ;FOLD F329 = T8 ;%{SE}%MKUKATPVW %CVW_SPS %VBOASG %P 2:F329 = T8, 3: BOASG
         $FLAG[329] = $TIMER_FLAG[8]
      ;ENDFOLD
      ;FOLD -- MS2 Reinigung beenden -- ;%{SE}%MKUKATPVW %CVW_COM %VCOMMENT %P 2:-- MS2 Reinigung beenden --, 3: VW_COMMENT
      ;ENDFOLD
      ;FOLD A1896 = AUS ;%{SE}%MKUKATPVW %CVW_SPS %VBOASG %P 2:A1896 = AUS, 3: BOASG
         $OUT[1896] = FALSE
      ;ENDFOLD
      ;FOLD -- MS2 Ausblasen AUS -- ;%{SE}%MKUKATPVW %CVW_COM %VCOMMENT %P 2:-- MS2 Ausblasen AUS --, 3: VW_COMMENT
      ;ENDFOLD
      ;FOLD A1902 = AUS ;%{SE}%MKUKATPVW %CVW_SPS %VBOASG %P 2:A1902 = AUS, 3: BOASG
         $OUT[1902] = FALSE
      ;ENDFOLD
      ;FOLD -- MS2 Einspruehen EIN -- ;%{SE}%MKUKATPVW %CVW_COM %VCOMMENT %P 2:-- MS2 Einspruehen EIN --, 3: VW_COMMENT
      ;ENDFOLD
      ;FOLD A528 = !F583 & F584 ;%{SE}%MKUKATPVW %CVW_SPS %VBOASG %P 2:A528 = !F583 & F584, 3: BOASG
         $OUT[528] = NOT $FLAG[583] AND $FLAG[584]
      ;ENDFOLD
      ;FOLD A1903 = F583 & F584 ;%{SE}%MKUKATPVW %CVW_SPS %VBOASG %P 2:A1903 = F583 & F584, 3: BOASG
         $OUT[1903] = $FLAG[583] AND $FLAG[584]
      ;ENDFOLD
      ;FOLD -- Einschaltdauer Einspruehen -- ;%{SE}%MKUKATPVW %CVW_COM %VCOMMENT %P 2:-- Einschaltdauer Einspruehen --, 3: VW_COMMENT
      ;ENDFOLD
      ;FOLD t7 ( EIN ) = i23[1/10Sek] ;%{SE}%MKUKATPVW %CVW_SPS %VTASG %P 2:t7 ( EIN ) = i23[1/10Sek], 3: TASG
         VW(#SET_TIME,TRUE,7,0,$COUNT_I[23])
      ;ENDFOLD
      ;FOLD Schritt 178 = A4039 ;%{SE}%MKUKATPVW %CVW_SPS %VST_CON %P 2:Schritt 178 = A4039, 3: ST_CON
         IF $OUT[4039] THEN
            PREVSTEP = $APP_INT[5]
            $APP_INT[5] = 178
         ENDIF
      ;ENDFOLD
   ;ENDFOLD
   ;FOLD SCHRITT 178 --MS2 Reinigung (an Pneum. Schwenkeinheit MS2)-- ;%{P}%MKUKATPVW,%CSTEP,%VST_NR,%P 1:SCHRITT, 2:178, 3:MS2 Reinigung (an Pneum. Schwenkeinheit MS2)
      ;FOLD ;%{H}
         Case 178
      ;ENDFOLD
      ;FOLD F323 = AUS ;%{SE}%MKUKATPVW %CVW_SPS %VBOASG %P 2:F323 = AUS, 3: BOASG
         $FLAG[323] = FALSE
      ;ENDFOLD
      ;FOLD A2171 = AUS ;%{SE}%MKUKATPVW %CVW_SPS %VBOASG %P 2:A2171 = AUS, 3: BOASG
         $OUT[2171] = FALSE
      ;ENDFOLD
      ;FOLD A2172 = AUS ;%{SE}%MKUKATPVW %CVW_SPS %VBOASG %P 2:A2172 = AUS, 3: BOASG
         $OUT[2172] = FALSE
      ;ENDFOLD
      ;FOLD A2173 = AUS ;%{SE}%MKUKATPVW %CVW_SPS %VBOASG %P 2:A2173 = AUS, 3: BOASG
         $OUT[2173] = FALSE
      ;ENDFOLD
      ;FOLD A2174 = AUS ;%{SE}%MKUKATPVW %CVW_SPS %VBOASG %P 2:A2174 = AUS, 3: BOASG
         $OUT[2174] = FALSE
      ;ENDFOLD
      ;FOLD A2175 = AUS ;%{SE}%MKUKATPVW %CVW_SPS %VBOASG %P 2:A2175 = AUS, 3: BOASG
         $OUT[2175] = FALSE
      ;ENDFOLD
      ;FOLD -- Ueberwachungszeit Schwenkeinheit 2 schwenken -- ;%{SE}%MKUKATPVW %CVW_COM %VCOMMENT %P 2:-- Ueberwachungszeit Schwenkeinheit 2 schwenken --, 3: VW_COMMENT
      ;ENDFOLD
      ;FOLD t8 ( EIN ) = -100[1/10Sek] ;%{SE}%MKUKATPVW %CVW_SPS %VTASG %P 2:t8 ( EIN ) = -100[1/10Sek], 3: TASG
         VW(#SET_TIME,TRUE,8,0,-100)
      ;ENDFOLD
      ;FOLD Schritt 179 = T7 & A4039 ;%{SE}%MKUKATPVW %CVW_SPS %VST_CON %P 2:Schritt 179 = T7 & A4039, 3: ST_CON
         IF $TIMER_FLAG[7] AND $OUT[4039] THEN
            PREVSTEP = $APP_INT[5]
            $APP_INT[5] = 179
         ENDIF
      ;ENDFOLD
   ;ENDFOLD
   ;FOLD SCHRITT 179 --MS2 Reinigung (an Pneum. Schwenkeinheit MS2)-- ;%{P}%MKUKATPVW,%CSTEP,%VST_NR,%P 1:SCHRITT, 2:179, 3:MS2 Reinigung (an Pneum. Schwenkeinheit MS2)
      ;FOLD ;%{H}
         Case 179
      ;ENDFOLD
      ;FOLD -- Steuerluft EIN -- ;%{SE}%MKUKATPVW %CVW_COM %VCOMMENT %P 2:-- Steuerluft EIN --, 3: VW_COMMENT
      ;ENDFOLD
      ;FOLD A2169 = A4039 ;%{SE}%MKUKATPVW %CVW_SPS %VBOASG %P 2:A2169 = A4039, 3: BOASG
         $OUT[2169] = $OUT[4039]
      ;ENDFOLD
      ;FOLD -- MS2 Einspruehen AUS -- ;%{SE}%MKUKATPVW %CVW_COM %VCOMMENT %P 2:-- MS2 Einspruehen AUS --, 3: VW_COMMENT
      ;ENDFOLD
      ;FOLD A528 = AUS ;%{SE}%MKUKATPVW %CVW_SPS %VBOASG %P 2:A528 = AUS, 3: BOASG
         $OUT[528] = FALSE
      ;ENDFOLD
      ;FOLD A1903 = AUS ;%{SE}%MKUKATPVW %CVW_SPS %VBOASG %P 2:A1903 = AUS, 3: BOASG
         $OUT[1903] = FALSE
      ;ENDFOLD
      ;FOLD -- Versetzeinheit in Ruhest. schw. -- ;%{SE}%MKUKATPVW %CVW_COM %VCOMMENT %P 2:-- Versetzeinheit in Ruhest. schw. --, 3: VW_COMMENT
      ;ENDFOLD
      ;FOLD A2175 = EIN ;%{SE}%MKUKATPVW %CVW_SPS %VBOASG %P 2:A2175 = EIN, 3: BOASG
         $OUT[2175] = TRUE
      ;ENDFOLD
      ;FOLD A2176 = AUS ;%{SE}%MKUKATPVW %CVW_SPS %VBOASG %P 2:A2176 = AUS, 3: BOASG
         $OUT[2176] = FALSE
      ;ENDFOLD
      ;FOLD -- RSK Fehlerausgabe Versetzeinheit in Ruhest. schw. -- ;%{SE}%MKUKATPVW %CVW_COM %VCOMMENT %P 2:-- RSK Fehlerausgabe Versetzeinheit in Ruhest. schw. --, 3: VW_COMMENT
      ;ENDFOLD
      ;FOLD F328 = F585 & T8 ;%{SE}%MKUKATPVW %CVW_SPS %VBOASG %P 2:F328 = F585 & T8, 3: BOASG
         $FLAG[328] = $FLAG[585] AND $TIMER_FLAG[8]
      ;ENDFOLD
      ;FOLD -- RSK Fehlerausgabe Schwenkeinheit 2 Arbeit. -- ;%{SE}%MKUKATPVW %CVW_COM %VCOMMENT %P 2:-- RSK Fehlerausgabe Schwenkeinheit 2 Arbeit. --, 3: VW_COMMENT
      ;ENDFOLD
      ;FOLD F324 = !E2172 & T8 ;%{SE}%MKUKATPVW %CVW_SPS %VBOASG %P 2:F324 = !E2172 & T8, 3: BOASG
         $FLAG[324] = NOT $IN[2172] AND $TIMER_FLAG[8]
      ;ENDFOLD
      ;FOLD -- RSK Sammelstoerung -- ;%{SE}%MKUKATPVW %CVW_COM %VCOMMENT %P 2:-- RSK Sammelstoerung --, 3: VW_COMMENT
      ;ENDFOLD
      ;FOLD F329 = F324 + F328 ;%{SE}%MKUKATPVW %CVW_SPS %VBOASG %P 2:F329 = F324 + F328, 3: BOASG
         $FLAG[329] = $FLAG[324] OR $FLAG[328]
      ;ENDFOLD
      ;FOLD Schritt 178 = (E26 + E27) & (F324 + F328) & A4039 ;%{SE}%MKUKATPVW %CVW_SPS %VST_CON %P 2:Schritt 178 = (E26 + E27) & (F324 + F328) & A4039, 3: ST_CON
         IF ($IN[26] OR $IN[27]) AND ($FLAG[324] OR $FLAG[328]) AND $OUT[4039] THEN
            PREVSTEP = $APP_INT[5]
            $APP_INT[5] = 178
         ENDIF
      ;ENDFOLD
      ;FOLD Schritt 180 = (!F324 + T8) & (F523 & !F524 & E2169 + !F523 & F524 & !E2170) & E2175 & F585 & A4039 ;%{SE}%MKUKATPVW %CVW_SPS %VST_CON %P 2:Schritt 180 = (!F324 + T8) & (F523 & !F524 & E2169 + !F523 & F524 & !E2170) & E2175 & F585 & A4039, 3: ST_CON
         IF (NOT $FLAG[324] OR $TIMER_FLAG[8]) AND ($FLAG[523] AND NOT $FLAG[524] AND $IN[2169] OR NOT $FLAG[523] AND $FLAG[524] AND NOT $IN[2170]) AND $IN[2175] AND $FLAG[585] AND $OUT[4039] THEN
            PREVSTEP = $APP_INT[5]
            $APP_INT[5] = 180
         ENDIF
      ;ENDFOLD
      ;FOLD Schritt 180 = (!F324 + T8) & (F523 & !F524 & E2169 + !F523 & F524 & !E2170) & !E2175 & !F585 & A4039 ;%{SE}%MKUKATPVW %CVW_SPS %VST_CON %P 2:Schritt 180 = (!F324 + T8) & (F523 & !F524 & E2169 + !F523 & F524 & !E2170) & !E2175 & !F585 & A4039, 3: ST_CON
         IF (NOT $FLAG[324] OR $TIMER_FLAG[8]) AND ($FLAG[523] AND NOT $FLAG[524] AND $IN[2169] OR NOT $FLAG[523] AND $FLAG[524] AND NOT $IN[2170]) AND NOT $IN[2175] AND NOT $FLAG[585] AND $OUT[4039] THEN
            PREVSTEP = $APP_INT[5]
            $APP_INT[5] = 180
         ENDIF
      ;ENDFOLD
   ;ENDFOLD
   ;FOLD SCHRITT 180 --MS2 Reinigung (an Pneum. Schwenkeinheit MS2)-- ;%{P}%MKUKATPVW,%CSTEP,%VST_NR,%P 1:SCHRITT, 2:180, 3:MS2 Reinigung (an Pneum. Schwenkeinheit MS2)
      ;FOLD ;%{H}
         Case 180
      ;ENDFOLD
      ;FOLD -- Steuerluft EIN -- ;%{SE}%MKUKATPVW %CVW_COM %VCOMMENT %P 2:-- Steuerluft EIN --, 3: VW_COMMENT
      ;ENDFOLD
      ;FOLD A2169 = A4039 ;%{SE}%MKUKATPVW %CVW_SPS %VBOASG %P 2:A2169 = A4039, 3: BOASG
         $OUT[2169] = $OUT[4039]
      ;ENDFOLD
      ;FOLD A2176 = AUS ;%{SE}%MKUKATPVW %CVW_SPS %VBOASG %P 2:A2176 = AUS, 3: BOASG
         $OUT[2176] = FALSE
      ;ENDFOLD
      ;FOLD -- Schwenkeinheit 2 in Ruhestellung schwenken -- ;%{SE}%MKUKATPVW %CVW_COM %VCOMMENT %P 2:-- Schwenkeinheit 2 in Ruhestellung schwenken --, 3: VW_COMMENT
      ;ENDFOLD
      ;FOLD A2171 = !E2171 ;%{SE}%MKUKATPVW %CVW_SPS %VBOASG %P 2:A2171 = !E2171, 3: BOASG
         $OUT[2171] = NOT $IN[2171]
      ;ENDFOLD
      ;FOLD A2172 = AUS ;%{SE}%MKUKATPVW %CVW_SPS %VBOASG %P 2:A2172 = AUS, 3: BOASG
         $OUT[2172] = FALSE
      ;ENDFOLD
      ;FOLD -- FRG Bewegung EIN -- ;%{SE}%MKUKATPVW %CVW_COM %VCOMMENT %P 2:-- FRG Bewegung EIN --, 3: VW_COMMENT
      ;ENDFOLD
      ;FOLD A2173 = AUS ;%{SE}%MKUKATPVW %CVW_SPS %VBOASG %P 2:A2173 = AUS, 3: BOASG
         $OUT[2173] = FALSE
      ;ENDFOLD
      ;FOLD A2174 = !E2171 ;%{SE}%MKUKATPVW %CVW_SPS %VBOASG %P 2:A2174 = !E2171, 3: BOASG
         $OUT[2174] = NOT $IN[2171]
      ;ENDFOLD
      ;FOLD Schritt 181 = E1896 & !E2172 & E2171 & A4039  + T8 ;%{SE}%MKUKATPVW %CVW_SPS %VST_CON %P 2:Schritt 181 = E1896 & !E2172 & E2171 & A4039  + T8, 3: ST_CON
